LIN {X 101.722,Y -39.308,Z -42.456,A -90.000,B 90.000,C 0.000} C_DIS
LIN {X 102.625,Y -39.308,Z -41.468,A -90.000,B 90.000,C 0.000} C_DIS
LIN {X 103.587,Y -39.308,Z -40.444,A -90.000,B 90.000,C 0.000} C_DIS
LIN {X 104.451,Y -39.308,Z -39.577,A -90.000,B 90.000,C 0.000} C_DIS
LIN {X 104.780,Y -39.308,Z -39.269,A -90.000,B 90.000,C 0.000} C_DIS
LIN {X 105.201,Y -39.308,Z -38.850,A -90.000,B 90.000,C 0.000} C_DIS
LIN {X 105.598,Y -39.308,Z -38.492,A -90.000,B 90.000,C 0.000} C_DIS
LIN {X 106.174,Y -39.308,Z -37.998,A -90.000,B 90.000,C 0.000} C_DIS
LIN {X 106.785,Y -39.308,Z -37.546,A -90.000,B 90.000,C 0.000} C_DIS
LIN {X 107.016,Y -39.308,Z -37.381,A -90.000,B 90.000,C 0.000} C_DIS
LIN {X 107.121,Y -39.308,Z -37.313,A -90.000,B 90.000,C 0.000} C_DIS
LIN {X 107.510,Y -39.308,Z -37.082,A -90.000,B 90.000,C 0.000} C_DIS
LIN {X 107.952,Y -39.308,Z -36.851,A -90.000,B 90.000,C 0.000} C_DIS
LIN {X 108.136,Y -39.308,Z -36.762,A -90.000,B 90.000,C 0.000} C_DIS
LIN {X 108.391,Y -39.308,Z -36.644,A -90.000,B 90.000,C 0.000} C_DIS
LIN {X 109.204,Y -39.308,Z -36.354,A -90.000,B 90.000,C 0.000} C_DIS
LIN {X 109.672,Y -39.308,Z -36.239,A -90.000,B 90.000,C 0.000} C_DIS
LIN {X 109.904,Y -39.308,Z -36.196,A -90.000,B 90.000,C 0.000} C_DIS
LIN {X 110.509,Y -39.308,Z -36.111,A -90.000,B 90.000,C 0.000} C_DIS
LIN {X 110.992,Y -39.308,Z -36.094,A -90.000,B 90.000,C 0.000} C_DIS
LIN {X 111.151,Y -39.308,Z -36.098,A -90.000,B 90.000,C 0.000} C_DIS
LIN {X 111.344,Y -39.308,Z -36.107,A -90.000,B 90.000,C 0.000} C_DIS
LIN {X 111.775,Y -39.308,Z -36.137,A -90.000,B 90.000,C 0.000} C_DIS
LIN {X 112.250,Y -39.308,Z -36.219,A -90.000,B 90.000,C 0.000} C_DIS
LIN {X 112.476,Y -39.308,Z -36.273,A -90.000,B 90.000,C 0.000} C_DIS
LIN {X 112.642,Y -39.308,Z -36.317,A -90.000,B 90.000,C 0.000} C_DIS
LIN {X 112.938,Y -39.308,Z -36.401,A -90.000,B 90.000,C 0.000} C_DIS
LIN {X 113.127,Y -39.308,Z -36.468,A -90.000,B 90.000,C 0.000} C_DIS
LIN {X 113.176,Y -39.308,Z -36.483,A -90.000,B 90.000,C 0.000} C_DIS
LIN {X 113.621,Y -39.308,Z -36.653,A -90.000,B 90.000,C 0.000} C_DIS
LIN {X 113.933,Y -39.308,Z -36.809,A -90.000,B 90.000,C 0.000} C_DIS
LIN {X 114.096,Y -39.308,Z -36.887,A -90.000,B 90.000,C 0.000} C_DIS
LIN {X 114.199,Y -39.308,Z -36.943,A -90.000,B 90.000,C 0.000} C_DIS
LIN {X 114.406,Y -39.308,Z -37.049,A -90.000,B 90.000,C 0.000} C_DIS
LIN {X 114.803,Y -39.308,Z -37.294,A -90.000,B 90.000,C 0.000} C_DIS
LIN {X 115.172,Y -39.308,Z -37.581,A -90.000,B 90.000,C 0.000} C_DIS
LIN {X 115.508,Y -39.308,Z -37.906,A -90.000,B 90.000,C 0.000} C_DIS
LIN {X 115.807,Y -39.308,Z -38.265,A -90.000,B 90.000,C 0.000} C_DIS
LIN {X 116.012,Y -39.308,Z -38.542,A -90.000,B 90.000,C 0.000} C_DIS
LIN {X 116.272,Y -39.308,Z -38.931,A -90.000,B 90.000,C 0.000} C_DIS
LIN {X 116.488,Y -39.308,Z -39.345,A -90.000,B 90.000,C 0.000} C_DIS
LIN {X 116.814,Y -39.308,Z -40.176,A -90.000,B 90.000,C 0.000} C_DIS
LIN {X 116.939,Y -39.308,Z -40.634,A -90.000,B 90.000,C 0.000} C_DIS
LIN {X 117.006,Y -39.308,Z -40.932,A -90.000,B 90.000,C 0.000} C_DIS
LIN {X 117.081,Y -39.308,Z -41.395,A -90.000,B 90.000,C 0.000} C_DIS
LIN {X 117.103,Y -39.308,Z -41.641,A -90.000,B 90.000,C 0.000} C_DIS
LIN {X 117.128,Y -39.308,Z -42.111,A -90.000,B 90.000,C 0.000} C_DIS
LIN {X 117.128,Y -39.308,Z -42.230,A -90.000,B 90.000,C 0.000} C_DIS
LIN {X 117.115,Y -39.308,Z -42.566,A -90.000,B 90.000,C 0.000} C_DIS
LIN {X 117.020,Y -39.308,Z -43.281,A -90.000,B 90.000,C 0.000} C_DIS
LIN {X 116.910,Y -39.308,Z -43.735,A -90.000,B 90.000,C 0.000} C_DIS
LIN {X 116.846,Y -39.308,Z -43.965,A -90.000,B 90.000,C 0.000} C_DIS
LIN {X 116.721,Y -39.308,Z -44.363,A -90.000,B 90.000,C 0.000} C_DIS
LIN {X 116.671,Y -39.308,Z -44.527,A -90.000,B 90.000,C 0.000} C_DIS
LIN {X 116.543,Y -39.308,Z -44.969,A -90.000,B 90.000,C 0.000} C_DIS
LIN {X 116.287,Y -39.308,Z -45.797,A -90.000,B 90.000,C 0.000} C_DIS
LIN {X 116.068,Y -39.308,Z -46.437,A -90.000,B 90.000,C 0.000} C_DIS
LIN {X 115.942,Y -39.308,Z -46.787,A -90.000,B 90.000,C 0.000} C_DIS
LIN {X 115.595,Y -39.308,Z -47.692,A -90.000,B 90.000,C 0.000} C_DIS
LIN {X 115.490,Y -39.308,Z -47.931,A -90.000,B 90.000,C 0.000} C_DIS
LIN {X 115.109,Y -39.308,Z -48.763,A -90.000,B 90.000,C 0.000} C_DIS
LIN {X 114.640,Y -39.308,Z -49.738,A -90.000,B 90.000,C 0.000} C_DIS
LIN {X 114.310,Y -39.308,Z -50.406,A -90.000,B 90.000,C 0.000} C_DIS
LIN {X 113.759,Y -39.308,Z -51.507,A -90.000,B 90.000,C 0.000} C_DIS
LIN {X 113.170,Y -39.308,Z -52.723,A -90.000,B 90.000,C 0.000} C_DIS
LIN {X 112.487,Y -39.308,Z -54.223,A -90.000,B 90.000,C 0.000} C_DIS
LIN {X 112.277,Y -39.308,Z -54.728,A -90.000,B 90.000,C 0.000} C_DIS
LIN {X 111.817,Y -39.308,Z -55.818,A -90.000,B 90.000,C 0.000} C_DIS
LIN {X 111.518,Y -39.308,Z -56.593,A -90.000,B 90.000,C 0.000} C_DIS
LIN {X 111.203,Y -39.308,Z -57.396,A -90.000,B 90.000,C 0.000} C_DIS
LIN {X 110.924,Y -39.308,Z -58.174,A -90.000,B 90.000,C 0.000} C_DIS
LIN {X 110.658,Y -39.308,Z -58.905,A -90.000,B 90.000,C 0.000} C_DIS
LIN {X 109.994,Y -39.308,Z -60.877,A -90.000,B 90.000,C 0.000} C_DIS
LIN {X 109.296,Y -39.308,Z -62.984,A -90.000,B 90.000,C 0.000} C_DIS
LIN {X 108.534,Y -39.308,Z -65.215,A -90.000,B 90.000,C 0.000} C_DIS
LIN {X 107.818,Y -39.308,Z -67.178,A -90.000,B 90.000,C 0.000} C_DIS
LIN {X 107.521,Y -39.308,Z -67.986,A -90.000,B 90.000,C 0.000} C_DIS
LIN {X 106.574,Y -39.308,Z -70.314,A -90.000,B 90.000,C 0.000} C_DIS
LIN {X 106.354,Y -39.308,Z -70.809,A -90.000,B 90.000,C 0.000} C_DIS
LIN {X 105.509,Y -39.308,Z -72.687,A -90.000,B 90.000,C 0.000} C_DIS
LIN {X 105.305,Y -39.308,Z -73.108,A -90.000,B 90.000,C 0.000} C_DIS
LIN {X 104.664,Y -39.308,Z -74.413,A -90.000,B 90.000,C 0.000} C_DIS
LIN {X 104.177,Y -39.308,Z -75.400,A -90.000,B 90.000,C 0.000} C_DIS
LIN {X 103.035,Y -39.308,Z -77.509,A -90.000,B 90.000,C 0.000} C_DIS
LIN {X 102.762,Y -39.308,Z -77.959,A -90.000,B 90.000,C 0.000} C_DIS
LIN {X 102.514,Y -39.308,Z -78.356,A -90.000,B 90.000,C 0.000} C_DIS
LIN {X 101.738,Y -39.308,Z -79.581,A -90.000,B 90.000,C 0.000} C_DIS
LIN {X 101.385,Y -39.308,Z -80.081,A -90.000,B 90.000,C 0.000} C_DIS
LIN {X 100.588,Y -39.308,Z -81.180,A -90.000,B 90.000,C 0.000} C_DIS
LIN {X 100.385,Y -39.308,Z -81.459,A -90.000,B 90.000,C 0.000} C_DIS
LIN {X 99.790,Y -39.308,Z -82.216,A -90.000,B 90.000,C 0.000} C_DIS
LIN {X 99.306,Y -39.308,Z -82.840,A -90.000,B 90.000,C 0.000} C_DIS
LIN {X 99.040,Y -39.308,Z -83.162,A -90.000,B 90.000,C 0.000} C_DIS
LIN {X 98.410,Y -39.308,Z -83.929,A -90.000,B 90.000,C 0.000} C_DIS
LIN {X 98.289,Y -39.308,Z -84.069,A -90.000,B 90.000,C 0.000} C_DIS
LIN {X 97.421,Y -39.308,Z -85.030,A -90.000,B 90.000,C 0.000} C_DIS
LIN {X 96.998,Y -39.308,Z -85.453,A -90.000,B 90.000,C 0.000} C_DIS
LIN {X 96.306,Y -39.308,Z -86.108,A -90.000,B 90.000,C 0.000} C_DIS
LIN {X 96.127,Y -39.308,Z -86.274,A -90.000,B 90.000,C 0.000} C_DIS
LIN {X 95.588,Y -39.308,Z -86.759,A -90.000,B 90.000,C 0.000} C_DIS
LIN {X 94.996,Y -39.308,Z -87.295,A -90.000,B 90.000,C 0.000} C_DIS
LIN {X 94.639,Y -39.308,Z -87.627,A -90.000,B 90.000,C 0.000} C_DIS
LIN {X 94.383,Y -39.308,Z -87.833,A -90.000,B 90.000,C 0.000} C_DIS
LIN {X 94.053,Y -39.308,Z -88.118,A -90.000,B 90.000,C 0.000} C_DIS
LIN {X 93.745,Y -39.308,Z -88.370,A -90.000,B 90.000,C 0.000} C_DIS
LIN {X 93.562,Y -39.308,Z -88.554,A -90.000,B 90.000,C 0.000} C_DIS
LIN {X 93.370,Y -39.308,Z -88.839,A -90.000,B 90.000,C 0.000} C_DIS
LIN {X 93.332,Y -39.308,Z -88.909,A -90.000,B 90.000,C 0.000} C_DIS
LIN {X 93.219,Y -39.308,Z -89.185,A -90.000,B 90.000,C 0.000} C_DIS
LIN {X 93.090,Y -39.308,Z -89.585,A -90.000,B 90.000,C 0.000} C_DIS
LIN {X 92.874,Y -39.308,Z -90.727,A -90.000,B 90.000,C 0.000} C_DIS
LIN {X 92.802,Y -39.308,Z -91.038,A -90.000,B 90.000,C 0.000} C_DIS
LIN {X 92.618,Y -39.308,Z -92.389,A -90.000,B 90.000,C 0.000} C_DIS
LIN {X 92.595,Y -39.308,Z -92.544,A -90.000,B 90.000,C 0.000} C_DIS
LIN {X 92.499,Y -39.308,Z -93.287,A -90.000,B 90.000,C 0.000} C_DIS
LIN {X 92.352,Y -39.308,Z -94.370,A -90.000,B 90.000,C 0.000} C_DIS
LIN {X 92.295,Y -39.308,Z -94.744,A -90.000,B 90.000,C 0.000} C_DIS
LIN {X 92.054,Y -39.308,Z -96.144,A -90.000,B 90.000,C 0.000} C_DIS
LIN {X 91.937,Y -39.308,Z -96.559,A -90.000,B 90.000,C 0.000} C_DIS
LIN {X 91.815,Y -39.308,Z -96.959,A -90.000,B 90.000,C 0.000} C_DIS
LIN {X 91.618,Y -39.308,Z -97.654,A -90.000,B 90.000,C 0.000} C_DIS
LIN {X 91.465,Y -39.308,Z -98.026,A -90.000,B 90.000,C 0.000} C_DIS
LIN {X 91.067,Y -39.308,Z -98.874,A -90.000,B 90.000,C 0.000} C_DIS
LIN {X 90.869,Y -39.308,Z -99.224,A -90.000,B 90.000,C 0.000} C_DIS
LIN {X 90.401,Y -39.308,Z -99.888,A -90.000,B 90.000,C 0.000} C_DIS
LIN {X 89.790,Y -39.308,Z -100.675,A -90.000,B 90.000,C 0.000} C_DIS
LIN {X 89.275,Y -39.308,Z -101.469,A -90.000,B 90.000,C 0.000} C_DIS
LIN {X 88.799,Y -39.308,Z -102.371,A -90.000,B 90.000,C 0.000} C_DIS
LIN {X 88.475,Y -39.308,Z -103.161,A -90.000,B 90.000,C 0.000} C_DIS
LIN {X 88.332,Y -39.308,Z -103.810,A -90.000,B 90.000,C 0.000} C_DIS
LIN {X 88.359,Y -39.308,Z -104.371,A -90.000,B 90.000,C 0.000} C_DIS
LIN {X 88.567,Y -39.308,Z -105.406,A -90.000,B 90.000,C 0.000} C_DIS
LIN {X 88.806,Y -39.308,Z -106.627,A -90.000,B 90.000,C 0.000} C_DIS
LIN {X 88.934,Y -39.308,Z -108.256,A -90.000,B 90.000,C 0.000} C_DIS
LIN {X 88.949,Y -39.308,Z -108.491,A -90.000,B 90.000,C 0.000} C_DIS
LIN {X 88.942,Y -39.308,Z -108.668,A -90.000,B 90.000,C 0.000} C_DIS
LIN {X 88.800,Y -39.308,Z -110.495,A -90.000,B 90.000,C 0.000} C_DIS
LIN {X 88.774,Y -39.308,Z -110.765,A -90.000,B 90.000,C 0.000} C_DIS
LIN {X 88.667,Y -39.308,Z -111.550,A -90.000,B 90.000,C 0.000} C_DIS
LIN {X 88.430,Y -39.308,Z -112.947,A -90.000,B 90.000,C 0.000} C_DIS
LIN {X 88.207,Y -39.308,Z -114.211,A -90.000,B 90.000,C 0.000} C_DIS
LIN {X 87.996,Y -39.308,Z -115.227,A -90.000,B 90.000,C 0.000} C_DIS
LIN {X 87.956,Y -39.308,Z -115.438,A -90.000,B 90.000,C 0.000} C_DIS
LIN {X 87.638,Y -39.308,Z -117.389,A -90.000,B 90.000,C 0.000} C_DIS
LIN {X 87.573,Y -39.308,Z -118.816,A -90.000,B 90.000,C 0.000} C_DIS
LIN {X 87.557,Y -39.308,Z -119.381,A -90.000,B 90.000,C 0.000} C_DIS
LIN {X 87.603,Y -39.308,Z -120.775,A -90.000,B 90.000,C 0.000} C_DIS
LIN {X 87.657,Y -39.308,Z -121.429,A -90.000,B 90.000,C 0.000} C_DIS
LIN {X 87.731,Y -39.308,Z -122.583,A -90.000,B 90.000,C 0.000} C_DIS
LIN {X 87.800,Y -39.308,Z -123.097,A -90.000,B 90.000,C 0.000} C_DIS
LIN {X 87.825,Y -39.308,Z -123.409,A -90.000,B 90.000,C 0.000} C_DIS
LIN {X 87.876,Y -39.308,Z -124.655,A -90.000,B 90.000,C 0.000} C_DIS
LIN {X 87.918,Y -39.308,Z -125.034,A -90.000,B 90.000,C 0.000} C_DIS
LIN {X 87.941,Y -39.308,Z -125.333,A -90.000,B 90.000,C 0.000} C_DIS
LIN {X 87.951,Y -39.308,Z -125.837,A -90.000,B 90.000,C 0.000} C_DIS
LIN {X 87.901,Y -39.308,Z -127.285,A -90.000,B 90.000,C 0.000} C_DIS
LIN {X 87.877,Y -39.308,Z -127.831,A -90.000,B 90.000,C 0.000} C_DIS
LIN {X 87.851,Y -39.308,Z -128.184,A -90.000,B 90.000,C 0.000} C_DIS
LIN {X 87.757,Y -39.308,Z -129.307,A -90.000,B 90.000,C 0.000} C_DIS
LIN {X 87.684,Y -39.308,Z -130.314,A -90.000,B 90.000,C 0.000} C_DIS
LIN {X 87.557,Y -39.308,Z -131.579,A -90.000,B 90.000,C 0.000} C_DIS
LIN {X 87.475,Y -39.308,Z -132.714,A -90.000,B 90.000,C 0.000} C_DIS
LIN {X 87.343,Y -39.308,Z -134.110,A -90.000,B 90.000,C 0.000} C_DIS
LIN {X 87.221,Y -39.308,Z -135.777,A -90.000,B 90.000,C 0.000} C_DIS
LIN {X 87.144,Y -39.308,Z -137.172,A -90.000,B 90.000,C 0.000} C_DIS
LIN {X 87.005,Y -39.308,Z -139.170,A -90.000,B 90.000,C 0.000} C_DIS
LIN {X 86.928,Y -39.308,Z -140.602,A -90.000,B 90.000,C 0.000} C_DIS
LIN {X 86.747,Y -39.308,Z -142.945,A -90.000,B 90.000,C 0.000} C_DIS
LIN {X 86.662,Y -39.308,Z -144.278,A -90.000,B 90.000,C 0.000} C_DIS
LIN {X 86.407,Y -39.308,Z -146.950,A -90.000,B 90.000,C 0.000} C_DIS
LIN {X 86.303,Y -39.308,Z -148.174,A -90.000,B 90.000,C 0.000} C_DIS
LIN {X 86.278,Y -39.308,Z -148.428,A -90.000,B 90.000,C 0.000} C_DIS
LIN {X 86.171,Y -39.308,Z -149.383,A -90.000,B 90.000,C 0.000} C_DIS
LIN {X 85.816,Y -39.308,Z -152.222,A -90.000,B 90.000,C 0.000} C_DIS
LIN {X 85.710,Y -39.308,Z -152.942,A -90.000,B 90.000,C 0.000} C_DIS
LIN {X 85.232,Y -39.308,Z -155.979,A -90.000,B 90.000,C 0.000} C_DIS
LIN {X 85.136,Y -39.308,Z -156.498,A -90.000,B 90.000,C 0.000} C_DIS
LIN {X 84.520,Y -39.308,Z -159.679,A -90.000,B 90.000,C 0.000} C_DIS
LIN {X 84.432,Y -39.308,Z -160.063,A -90.000,B 90.000,C 0.000} C_DIS
LIN {X 83.664,Y -39.308,Z -163.335,A -90.000,B 90.000,C 0.000} C_DIS
LIN {X 83.589,Y -39.308,Z -163.643,A -90.000,B 90.000,C 0.000} C_DIS
LIN {X 82.601,Y -39.308,Z -167.169,A -90.000,B 90.000,C 0.000} C_DIS
LIN {X 81.544,Y -39.308,Z -170.573,A -90.000,B 90.000,C 0.000} C_DIS
LIN {X 80.492,Y -39.308,Z -173.831,A -90.000,B 90.000,C 0.000} C_DIS
LIN {X 80.289,Y -39.308,Z -174.485,A -90.000,B 90.000,C 0.000} C_DIS
LIN {X 79.518,Y -39.308,Z -176.924,A -90.000,B 90.000,C 0.000} C_DIS
LIN {X 78.896,Y -39.308,Z -179.083,A -90.000,B 90.000,C 0.000} C_DIS
LIN {X 78.733,Y -39.308,Z -179.680,A -90.000,B 90.000,C 0.000} C_DIS
LIN {X 78.239,Y -39.308,Z -181.531,A -90.000,B 90.000,C 0.000} C_DIS
LIN {X 78.020,Y -39.308,Z -182.417,A -90.000,B 90.000,C 0.000} C_DIS
LIN {X 77.515,Y -39.308,Z -184.388,A -90.000,B 90.000,C 0.000} C_DIS
LIN {X 77.360,Y -39.308,Z -185.055,A -90.000,B 90.000,C 0.000} C_DIS
LIN {X 76.824,Y -39.308,Z -187.147,A -90.000,B 90.000,C 0.000} C_DIS
LIN {X 76.720,Y -39.308,Z -187.594,A -90.000,B 90.000,C 0.000} C_DIS
LIN {X 76.130,Y -39.308,Z -189.797,A -90.000,B 90.000,C 0.000} C_DIS
LIN {X 76.066,Y -39.308,Z -190.059,A -90.000,B 90.000,C 0.000} C_DIS
LIN {X 75.356,Y -39.308,Z -192.504,A -90.000,B 90.000,C 0.000} C_DIS
LIN {X 75.319,Y -39.308,Z -192.641,A -90.000,B 90.000,C 0.000} C_DIS
LIN {X 75.217,Y -39.308,Z -192.988,A -90.000,B 90.000,C 0.000} C_DIS
LIN {X 74.311,Y -39.308,Z -195.828,A -90.000,B 90.000,C 0.000} C_DIS
LIN {X 73.163,Y -39.308,Z -199.116,A -90.000,B 90.000,C 0.000} C_DIS
LIN {X 71.708,Y -39.308,Z -203.024,A -90.000,B 90.000,C 0.000} C_DIS
LIN {X 69.982,Y -39.308,Z -207.432,A -90.000,B 90.000,C 0.000} C_DIS
LIN {X 67.893,Y -39.308,Z -212.535,A -90.000,B 90.000,C 0.000} C_DIS
LIN {X 66.291,Y -39.308,Z -216.289,A -90.000,B 90.000,C 0.000} C_DIS
LIN {X 65.715,Y -39.308,Z -217.628,A -90.000,B 90.000,C 0.000} C_DIS
LIN {X 63.402,Y -39.308,Z -222.773,A -90.000,B 90.000,C 0.000} C_DIS
LIN {X 60.817,Y -39.308,Z -228.203,A -90.000,B 90.000,C 0.000} C_DIS
LIN {X 58.290,Y -39.308,Z -233.168,A -90.000,B 90.000,C 0.000} C_DIS
LIN {X 58.161,Y -39.308,Z -233.430,A -90.000,B 90.000,C 0.000} C_DIS
LIN {X 58.084,Y -39.308,Z -233.572,A -90.000,B 90.000,C 0.000} C_DIS
LIN {X 55.501,Y -39.308,Z -238.273,A -90.000,B 90.000,C 0.000} C_DIS
LIN {X 55.234,Y -39.308,Z -238.790,A -90.000,B 90.000,C 0.000} C_DIS
LIN {X 54.905,Y -39.308,Z -239.394,A -90.000,B 90.000,C 0.000} C_DIS
LIN {X 54.713,Y -39.308,Z -239.734,A -90.000,B 90.000,C 0.000} C_DIS
LIN {X 52.416,Y -39.308,Z -243.561,A -90.000,B 90.000,C 0.000} C_DIS
LIN {X 52.416,Y -60.000,Z -243.561,A -90.000,B 90.000,C 0.000} C_DIS
LIN {X 101.612,Y -60.000,Z -42.574,A -90.000,B 90.000,C 0.000} C_DIS
LIN {X 101.612,Y -37.308,Z -42.574,A -90.000,B 90.000,C 0.000} C_DIS
LIN {X 101.629,Y -37.311,Z -42.419,A -90.000,B 90.000,C 0.000} C_DIS
LIN {X 101.656,Y -37.315,Z -42.297,A -90.000,B 90.000,C 0.000} C_DIS
LIN {X 101.723,Y -37.329,Z -42.033,A -90.000,B 90.000,C 0.000} C_DIS
LIN {X 101.775,Y -37.337,Z -41.902,A -90.000,B 90.000,C 0.000} C_DIS
LIN {X 101.877,Y -37.355,Z -41.654,A -90.000,B 90.000,C 0.000} C_DIS
LIN {X 102.047,Y -37.380,Z -41.312,A -90.000,B 90.000,C 0.000} C_DIS
LIN {X 102.134,Y -37.395,Z -41.144,A -90.000,B 90.000,C 0.000} C_DIS
LIN {X 102.399,Y -37.434,Z -40.690,A -90.000,B 90.000,C 0.000} C_DIS
LIN {X 102.645,Y -37.468,Z -40.302,A -90.000,B 90.000,C 0.000} C_DIS
LIN {X 102.898,Y -37.488,Z -39.967,A -90.000,B 90.000,C 0.000} C_DIS
LIN {X 103.145,Y -37.508,Z -39.654,A -90.000,B 90.000,C 0.000} C_DIS
LIN {X 103.251,Y -37.517,Z -39.521,A -90.000,B 90.000,C 0.000} C_DIS
LIN {X 103.626,Y -37.529,Z -39.112,A -90.000,B 90.000,C 0.000} C_DIS
LIN {X 103.738,Y -37.531,Z -38.993,A -90.000,B 90.000,C 0.000} C_DIS
LIN {X 103.970,Y -37.536,Z -38.759,A -90.000,B 90.000,C 0.000} C_DIS
LIN {X 104.139,Y -37.537,Z -38.598,A -90.000,B 90.000,C 0.000} C_DIS
LIN {X 104.427,Y -37.532,Z -38.323,A -90.000,B 90.000,C 0.000} C_DIS
LIN {X 104.582,Y -37.527,Z -38.183,A -90.000,B 90.000,C 0.000} C_DIS
LIN {X 104.958,Y -37.514,Z -37.880,A -90.000,B 90.000,C 0.000} C_DIS
LIN {X 105.114,Y -37.508,Z -37.759,A -90.000,B 90.000,C 0.000} C_DIS
LIN {X 105.454,Y -37.493,Z -37.511,A -90.000,B 90.000,C 0.000} C_DIS
LIN {X 105.665,Y -37.480,Z -37.367,A -90.000,B 90.000,C 0.000} C_DIS
LIN {X 105.896,Y -37.473,Z -37.215,A -90.000,B 90.000,C 0.000} C_DIS
LIN {X 106.119,Y -37.463,Z -37.081,A -90.000,B 90.000,C 0.000} C_DIS
LIN {X 106.362,Y -37.448,Z -36.944,A -90.000,B 90.000,C 0.000} C_DIS
LIN {X 106.738,Y -37.432,Z -36.736,A -90.000,B 90.000,C 0.000} C_DIS
LIN {X 106.867,Y -37.429,Z -36.668,A -90.000,B 90.000,C 0.000} C_DIS
LIN {X 106.984,Y -37.425,Z -36.612,A -90.000,B 90.000,C 0.000} C_DIS
LIN {X 107.278,Y -37.416,Z -36.473,A -90.000,B 90.000,C 0.000} C_DIS
LIN {X 107.430,Y -37.413,Z -36.403,A -90.000,B 90.000,C 0.000} C_DIS
LIN {X 107.770,Y -37.406,Z -36.252,A -90.000,B 90.000,C 0.000} C_DIS
LIN {X 108.143,Y -37.398,Z -36.107,A -90.000,B 90.000,C 0.000} C_DIS
LIN {X 108.234,Y -37.397,Z -36.075,A -90.000,B 90.000,C 0.000} C_DIS
LIN {X 108.294,Y -37.398,Z -36.051,A -90.000,B 90.000,C 0.000} C_DIS
LIN {X 109.071,Y -37.390,Z -35.804,A -90.000,B 90.000,C 0.000} C_DIS
LIN {X 109.166,Y -37.391,Z -35.777,A -90.000,B 90.000,C 0.000} C_DIS
LIN {X 109.380,Y -37.390,Z -35.728,A -90.000,B 90.000,C 0.000} C_DIS
LIN {X 109.499,Y -37.389,Z -35.704,A -90.000,B 90.000,C 0.000} C_DIS
LIN {X 109.570,Y -37.389,Z -35.688,A -90.000,B 90.000,C 0.000} C_DIS
LIN {X 109.857,Y -37.390,Z -35.632,A -90.000,B 90.000,C 0.000} C_DIS
LIN {X 110.012,Y -37.392,Z -35.602,A -90.000,B 90.000,C 0.000} C_DIS
LIN {X 110.069,Y -37.392,Z -35.595,A -90.000,B 90.000,C 0.000} C_DIS
LIN {X 110.465,Y -37.387,Z -35.558,A -90.000,B 90.000,C 0.000} C_DIS
LIN {X 111.003,Y -37.390,Z -35.530,A -90.000,B 90.000,C 0.000} C_DIS
LIN {X 111.317,Y -37.391,Z -35.537,A -90.000,B 90.000,C 0.000} C_DIS
LIN {X 111.666,Y -37.392,Z -35.557,A -90.000,B 90.000,C 0.000} C_DIS
LIN {X 111.823,Y -37.390,Z -35.574,A -90.000,B 90.000,C 0.000} C_DIS
LIN {X 112.066,Y -37.392,Z -35.605,A -90.000,B 90.000,C 0.000} C_DIS
LIN {X 112.386,Y -37.394,Z -35.655,A -90.000,B 90.000,C 0.000} C_DIS
LIN {X 112.546,Y -37.398,Z -35.681,A -90.000,B 90.000,C 0.000} C_DIS
LIN {X 112.867,Y -37.398,Z -35.764,A -90.000,B 90.000,C 0.000} C_DIS
LIN {X 113.101,Y -37.399,Z -35.828,A -90.000,B 90.000,C 0.000} C_DIS
LIN {X 113.182,Y -37.400,Z -35.851,A -90.000,B 90.000,C 0.000} C_DIS
LIN {X 113.401,Y -37.401,Z -35.926,A -90.000,B 90.000,C 0.000} C_DIS
LIN {X 113.848,Y -37.399,Z -36.104,A -90.000,B 90.000,C 0.000} C_DIS
LIN {X 114.023,Y -37.401,Z -36.180,A -90.000,B 90.000,C 0.000} C_DIS
LIN {X 114.165,Y -37.404,Z -36.241,A -90.000,B 90.000,C 0.000} C_DIS
LIN {X 114.592,Y -37.402,Z -36.465,A -90.000,B 90.000,C 0.000} C_DIS
LIN {X 114.656,Y -37.401,Z -36.500,A -90.000,B 90.000,C 0.000} C_DIS
LIN {X 115.108,Y -37.394,Z -36.801,A -90.000,B 90.000,C 0.000} C_DIS
LIN {X 115.164,Y -37.394,Z -36.841,A -90.000,B 90.000,C 0.000} C_DIS
LIN {X 115.527,Y -37.390,Z -37.143,A -90.000,B 90.000,C 0.000} C_DIS
LIN {X 115.726,Y -37.387,Z -37.344,A -90.000,B 90.000,C 0.000} C_DIS
LIN {X 115.932,Y -37.385,Z -37.557,A -90.000,B 90.000,C 0.000} C_DIS
LIN {X 116.140,Y -37.386,Z -37.800,A -90.000,B 90.000,C 0.000} C_DIS
LIN {X 116.249,Y -37.385,Z -37.938,A -90.000,B 90.000,C 0.000} C_DIS
LIN {X 116.441,Y -37.388,Z -38.181,A -90.000,B 90.000,C 0.000} C_DIS
LIN {X 116.702,Y -37.384,Z -38.591,A -90.000,B 90.000,C 0.000} C_DIS
LIN {X 116.836,Y -37.381,Z -38.860,A -90.000,B 90.000,C 0.000} C_DIS
LIN {X 116.930,Y -37.379,Z -39.049,A -90.000,B 90.000,C 0.000} C_DIS
LIN {X 116.972,Y -37.377,Z -39.155,A -90.000,B 90.000,C 0.000} C_DIS
LIN {X 117.070,Y -37.377,Z -39.405,A -90.000,B 90.000,C 0.000} C_DIS
LIN {X 117.242,Y -37.375,Z -39.860,A -90.000,B 90.000,C 0.000} C_DIS
LIN {X 117.288,Y -37.371,Z -40.034,A -90.000,B 90.000,C 0.000} C_DIS
LIN {X 117.365,Y -37.370,Z -40.328,A -90.000,B 90.000,C 0.000} C_DIS
LIN {X 117.387,Y -37.368,Z -40.432,A -90.000,B 90.000,C 0.000} C_DIS
LIN {X 117.421,Y -37.365,Z -40.627,A -90.000,B 90.000,C 0.000} C_DIS
LIN {X 117.443,Y -37.365,Z -40.728,A -90.000,B 90.000,C 0.000} C_DIS
LIN {X 117.518,Y -37.362,Z -41.208,A -90.000,B 90.000,C 0.000} C_DIS
LIN {X 117.529,Y -37.361,Z -41.323,A -90.000,B 90.000,C 0.000} C_DIS
LIN {X 117.541,Y -37.361,Z -41.406,A -90.000,B 90.000,C 0.000} C_DIS
LIN {X 117.552,Y -37.362,Z -41.518,A -90.000,B 90.000,C 0.000} C_DIS
LIN {X 117.566,Y -37.363,Z -41.618,A -90.000,B 90.000,C 0.000} C_DIS
LIN {X 117.582,Y -37.364,Z -41.824,A -90.000,B 90.000,C 0.000} C_DIS
LIN {X 117.598,Y -37.364,Z -42.113,A -90.000,B 90.000,C 0.000} C_DIS
LIN {X 117.615,Y -37.371,Z -42.456,A -90.000,B 90.000,C 0.000} C_DIS
LIN {X 117.612,Y -37.371,Z -42.585,A -90.000,B 90.000,C 0.000} C_DIS
LIN {X 117.603,Y -37.375,Z -42.769,A -90.000,B 90.000,C 0.000} C_DIS
LIN {X 117.568,Y -37.384,Z -43.280,A -90.000,B 90.000,C 0.000} C_DIS
LIN {X 117.546,Y -37.385,Z -43.434,A -90.000,B 90.000,C 0.000} C_DIS
LIN {X 117.522,Y -37.389,Z -43.592,A -90.000,B 90.000,C 0.000} C_DIS
LIN {X 117.495,Y -37.396,Z -43.809,A -90.000,B 90.000,C 0.000} C_DIS
LIN {X 117.421,Y -37.410,Z -44.234,A -90.000,B 90.000,C 0.000} C_DIS
LIN {X 117.382,Y -37.415,Z -44.407,A -90.000,B 90.000,C 0.000} C_DIS
LIN {X 117.286,Y -37.424,Z -44.814,A -90.000,B 90.000,C 0.000} C_DIS
LIN {X 117.193,Y -37.430,Z -45.193,A -90.000,B 90.000,C 0.000} C_DIS
LIN {X 117.168,Y -37.432,Z -45.287,A -90.000,B 90.000,C 0.000} C_DIS
LIN {X 116.978,Y -37.434,Z -45.926,A -90.000,B 90.000,C 0.000} C_DIS
LIN {X 116.921,Y -37.433,Z -46.095,A -90.000,B 90.000,C 0.000} C_DIS
LIN {X 116.602,Y -37.428,Z -46.967,A -90.000,B 90.000,C 0.000} C_DIS
LIN {X 116.539,Y -37.429,Z -47.137,A -90.000,B 90.000,C 0.000} C_DIS
LIN {X 116.189,Y -37.416,Z -47.952,A -90.000,B 90.000,C 0.000} C_DIS
LIN {X 116.156,Y -37.416,Z -48.026,A -90.000,B 90.000,C 0.000} C_DIS
LIN {X 115.889,Y -37.410,Z -48.572,A -90.000,B 90.000,C 0.000} C_DIS
LIN {X 115.501,Y -37.403,Z -49.350,A -90.000,B 90.000,C 0.000} C_DIS
LIN {X 115.430,Y -37.402,Z -49.492,A -90.000,B 90.000,C 0.000} C_DIS
LIN {X 114.861,Y -37.394,Z -50.596,A -90.000,B 90.000,C 0.000} C_DIS
LIN {X 114.199,Y -37.389,Z -51.887,A -90.000,B 90.000,C 0.000} C_DIS
LIN {X 113.591,Y -37.385,Z -53.125,A -90.000,B 90.000,C 0.000} C_DIS
LIN {X 113.530,Y -37.385,Z -53.256,A -90.000,B 90.000,C 0.000} C_DIS
LIN {X 113.048,Y -37.385,Z -54.319,A -90.000,B 90.000,C 0.000} C_DIS
LIN {X 112.975,Y -37.387,Z -54.492,A -90.000,B 90.000,C 0.000} C_DIS
LIN {X 112.392,Y -37.388,Z -55.887,A -90.000,B 90.000,C 0.000} C_DIS
LIN {X 111.753,Y -37.390,Z -57.546,A -90.000,B 90.000,C 0.000} C_DIS
LIN {X 111.203,Y -37.393,Z -59.096,A -90.000,B 90.000,C 0.000} C_DIS
LIN {X 110.557,Y -37.398,Z -61.065,A -90.000,B 90.000,C 0.000} C_DIS
LIN {X 109.947,Y -37.403,Z -62.950,A -90.000,B 90.000,C 0.000} C_DIS
LIN {X 109.226,Y -37.404,Z -65.082,A -90.000,B 90.000,C 0.000} C_DIS
LIN {X 108.967,Y -37.403,Z -65.799,A -90.000,B 90.000,C 0.000} C_DIS
LIN {X 108.309,Y -37.403,Z -67.604,A -90.000,B 90.000,C 0.000} C_DIS
LIN {X 108.225,Y -37.403,Z -67.833,A -90.000,B 90.000,C 0.000} C_DIS
LIN {X 108.076,Y -37.400,Z -68.212,A -90.000,B 90.000,C 0.000} C_DIS
LIN {X 107.446,Y -37.404,Z -69.796,A -90.000,B 90.000,C 0.000} C_DIS
LIN {X 107.263,Y -37.405,Z -70.252,A -90.000,B 90.000,C 0.000} C_DIS
LIN {X 107.131,Y -37.403,Z -70.562,A -90.000,B 90.000,C 0.000} C_DIS
LIN {X 106.480,Y -37.411,Z -72.071,A -90.000,B 90.000,C 0.000} C_DIS
LIN {X 106.196,Y -37.413,Z -72.716,A -90.000,B 90.000,C 0.000} C_DIS
LIN {X 105.877,Y -37.413,Z -73.388,A -90.000,B 90.000,C 0.000} C_DIS
LIN {X 105.250,Y -37.419,Z -74.707,A -90.000,B 90.000,C 0.000} C_DIS
LIN {X 105.072,Y -37.421,Z -75.080,A -90.000,B 90.000,C 0.000} C_DIS
LIN {X 104.900,Y -37.421,Z -75.429,A -90.000,B 90.000,C 0.000} C_DIS
LIN {X 104.753,Y -37.419,Z -75.712,A -90.000,B 90.000,C 0.000} C_DIS
LIN {X 104.386,Y -37.423,Z -76.414,A -90.000,B 90.000,C 0.000} C_DIS
LIN {X 103.785,Y -37.431,Z -77.572,A -90.000,B 90.000,C 0.000} C_DIS
LIN {X 103.595,Y -37.428,Z -77.899,A -90.000,B 90.000,C 0.000} C_DIS
LIN {X 103.168,Y -37.435,Z -78.630,A -90.000,B 90.000,C 0.000} C_DIS
LIN {X 102.802,Y -37.445,Z -79.256,A -90.000,B 90.000,C 0.000} C_DIS
LIN {X 102.670,Y -37.446,Z -79.472,A -90.000,B 90.000,C 0.000} C_DIS
LIN {X 102.431,Y -37.446,Z -79.850,A -90.000,B 90.000,C 0.000} C_DIS
LIN {X 102.263,Y -37.446,Z -80.100,A -90.000,B 90.000,C 0.000} C_DIS
LIN {X 101.641,Y -37.458,Z -81.020,A -90.000,B 90.000,C 0.000} C_DIS
LIN {X 101.342,Y -37.466,Z -81.465,A -90.000,B 90.000,C 0.000} C_DIS
LIN {X 100.998,Y -37.466,Z -81.940,A -90.000,B 90.000,C 0.000} C_DIS
LIN {X 100.316,Y -37.486,Z -82.881,A -90.000,B 90.000,C 0.000} C_DIS
LIN {X 99.946,Y -37.489,Z -83.371,A -90.000,B 90.000,C 0.000} C_DIS
LIN {X 99.578,Y -37.501,Z -83.856,A -90.000,B 90.000,C 0.000} C_DIS
LIN {X 99.261,Y -37.508,Z -84.264,A -90.000,B 90.000,C 0.000} C_DIS
LIN {X 99.033,Y -37.512,Z -84.555,A -90.000,B 90.000,C 0.000} C_DIS
LIN {X 98.364,Y -37.544,Z -85.391,A -90.000,B 90.000,C 0.000} C_DIS
LIN {X 98.095,Y -37.550,Z -85.703,A -90.000,B 90.000,C 0.000} C_DIS
LIN {X 97.667,Y -37.573,Z -86.186,A -90.000,B 90.000,C 0.000} C_DIS
LIN {X 97.025,Y -37.612,Z -86.887,A -90.000,B 90.000,C 0.000} C_DIS
LIN {X 96.296,Y -37.671,Z -87.668,A -90.000,B 90.000,C 0.000} C_DIS
LIN {X 96.049,Y -37.693,Z -87.933,A -90.000,B 90.000,C 0.000} C_DIS
LIN {X 95.768,Y -37.712,Z -88.223,A -90.000,B 90.000,C 0.000} C_DIS
LIN {X 95.527,Y -37.724,Z -88.468,A -90.000,B 90.000,C 0.000} C_DIS
LIN {X 95.414,Y -37.740,Z -88.596,A -90.000,B 90.000,C 0.000} C_DIS
LIN {X 95.283,Y -37.762,Z -88.737,A -90.000,B 90.000,C 0.000} C_DIS
LIN {X 95.137,Y -37.809,Z -88.930,A -90.000,B 90.000,C 0.000} C_DIS
LIN {X 95.057,Y -37.828,Z -89.028,A -90.000,B 90.000,C 0.000} C_DIS
LIN {X 94.951,Y -37.875,Z -89.185,A -90.000,B 90.000,C 0.000} C_DIS
LIN {X 94.862,Y -37.915,Z -89.309,A -90.000,B 90.000,C 0.000} C_DIS
LIN {X 94.745,Y -37.967,Z -89.468,A -90.000,B 90.000,C 0.000} C_DIS
LIN {X 94.719,Y -37.976,Z -89.506,A -90.000,B 90.000,C 0.000} C_DIS
LIN {X 94.678,Y -37.988,Z -89.586,A -90.000,B 90.000,C 0.000} C_DIS
LIN {X 94.654,Y -37.992,Z -89.654,A -90.000,B 90.000,C 0.000} C_DIS
LIN {X 94.638,Y -37.996,Z -89.703,A -90.000,B 90.000,C 0.000} C_DIS
LIN {X 94.564,Y -38.006,Z -89.961,A -90.000,B 90.000,C 0.000} C_DIS
LIN {X 94.501,Y -37.998,Z -90.254,A -90.000,B 90.000,C 0.000} C_DIS
LIN {X 94.353,Y -37.992,Z -91.007,A -90.000,B 90.000,C 0.000} C_DIS
LIN {X 94.290,Y -37.999,Z -91.311,A -90.000,B 90.000,C 0.000} C_DIS
LIN {X 94.101,Y -37.984,Z -92.611,A -90.000,B 90.000,C 0.000} C_DIS
LIN {X 94.070,Y -37.984,Z -92.818,A -90.000,B 90.000,C 0.000} C_DIS
LIN {X 93.913,Y -37.974,Z -93.948,A -90.000,B 90.000,C 0.000} C_DIS
LIN {X 93.822,Y -37.971,Z -94.588,A -90.000,B 90.000,C 0.000} C_DIS
LIN {X 93.755,Y -37.965,Z -94.995,A -90.000,B 90.000,C 0.000} C_DIS
LIN {X 93.555,Y -37.959,Z -96.126,A -90.000,B 90.000,C 0.000} C_DIS
LIN {X 93.490,Y -37.944,Z -96.420,A -90.000,B 90.000,C 0.000} C_DIS
LIN {X 93.467,Y -37.942,Z -96.514,A -90.000,B 90.000,C 0.000} C_DIS
LIN {X 93.333,Y -37.941,Z -96.985,A -90.000,B 90.000,C 0.000} C_DIS
LIN {X 93.225,Y -37.947,Z -97.360,A -90.000,B 90.000,C 0.000} C_DIS
LIN {X 93.161,Y -37.949,Z -97.590,A -90.000,B 90.000,C 0.000} C_DIS
LIN {X 93.065,Y -37.941,Z -97.900,A -90.000,B 90.000,C 0.000} C_DIS
LIN {X 93.052,Y -37.940,Z -97.943,A -90.000,B 90.000,C 0.000} C_DIS
LIN {X 92.986,Y -37.928,Z -98.127,A -90.000,B 90.000,C 0.000} C_DIS
LIN {X 92.880,Y -37.928,Z -98.391,A -90.000,B 90.000,C 0.000} C_DIS
LIN {X 92.777,Y -37.930,Z -98.642,A -90.000,B 90.000,C 0.000} C_DIS
LIN {X 92.700,Y -37.936,Z -98.819,A -90.000,B 90.000,C 0.000} C_DIS
LIN {X 92.504,Y -37.935,Z -99.235,A -90.000,B 90.000,C 0.000} C_DIS
LIN {X 92.382,Y -37.923,Z -99.469,A -90.000,B 90.000,C 0.000} C_DIS
LIN {X 92.331,Y -37.921,Z -99.562,A -90.000,B 90.000,C 0.000} C_DIS
LIN {X 92.130,Y -37.919,Z -99.915,A -90.000,B 90.000,C 0.000} C_DIS
LIN {X 92.056,Y -37.921,Z -100.038,A -90.000,B 90.000,C 0.000} C_DIS
LIN {X 91.988,Y -37.926,Z -100.144,A -90.000,B 90.000,C 0.000} C_DIS
LIN {X 91.563,Y -37.946,Z -100.779,A -90.000,B 90.000,C 0.000} C_DIS
LIN {X 91.542,Y -37.948,Z -100.808,A -90.000,B 90.000,C 0.000} C_DIS
LIN {X 91.031,Y -38.022,Z -101.576,A -90.000,B 90.000,C 0.000} C_DIS
LIN {X 91.015,Y -38.024,Z -101.602,A -90.000,B 90.000,C 0.000} C_DIS
LIN {X 90.639,Y -38.082,Z -102.269,A -90.000,B 90.000,C 0.000} C_DIS
LIN {X 90.473,Y -38.089,Z -102.595,A -90.000,B 90.000,C 0.000} C_DIS
LIN {X 90.261,Y -38.124,Z -103.054,A -90.000,B 90.000,C 0.000} C_DIS
LIN {X 90.095,Y -38.125,Z -103.461,A -90.000,B 90.000,C 0.000} C_DIS
LIN {X 90.030,Y -38.141,Z -103.648,A -90.000,B 90.000,C 0.000} C_DIS
LIN {X 89.963,Y -38.139,Z -103.948,A -90.000,B 90.000,C 0.000} C_DIS
LIN {X 89.956,Y -38.119,Z -104.102,A -90.000,B 90.000,C 0.000} C_DIS
LIN {X 89.958,Y -38.118,Z -104.173,A -90.000,B 90.000,C 0.000} C_DIS
LIN {X 90.011,Y -38.084,Z -104.566,A -90.000,B 90.000,C 0.000} C_DIS
LIN {X 90.205,Y -38.074,Z -105.581,A -90.000,B 90.000,C 0.000} C_DIS
LIN {X 90.351,Y -38.075,Z -106.324,A -90.000,B 90.000,C 0.000} C_DIS
LIN {X 90.382,Y -38.081,Z -106.521,A -90.000,B 90.000,C 0.000} C_DIS
LIN {X 90.412,Y -38.094,Z -106.777,A -90.000,B 90.000,C 0.000} C_DIS
LIN {X 90.513,Y -38.112,Z -107.883,A -90.000,B 90.000,C 0.000} C_DIS
LIN {X 90.549,Y -38.113,Z -108.383,A -90.000,B 90.000,C 0.000} C_DIS
LIN {X 90.554,Y -38.117,Z -108.554,A -90.000,B 90.000,C 0.000} C_DIS
LIN {X 90.554,Y -38.119,Z -108.593,A -90.000,B 90.000,C 0.000} C_DIS
LIN {X 90.545,Y -38.119,Z -108.793,A -90.000,B 90.000,C 0.000} C_DIS
LIN {X 90.514,Y -38.121,Z -109.211,A -90.000,B 90.000,C 0.000} C_DIS
LIN {X 90.436,Y -38.151,Z -110.490,A -90.000,B 90.000,C 0.000} C_DIS
LIN {X 90.425,Y -38.154,Z -110.656,A -90.000,B 90.000,C 0.000} C_DIS
LIN {X 90.389,Y -38.149,Z -110.985,A -90.000,B 90.000,C 0.000} C_DIS
LIN {X 90.325,Y -38.151,Z -111.461,A -90.000,B 90.000,C 0.000} C_DIS
LIN {X 90.280,Y -38.159,Z -111.825,A -90.000,B 90.000,C 0.000} C_DIS
LIN {X 90.145,Y -38.193,Z -112.761,A -90.000,B 90.000,C 0.000} C_DIS
LIN {X 89.990,Y -38.208,Z -113.716,A -90.000,B 90.000,C 0.000} C_DIS
LIN {X 89.859,Y -38.235,Z -114.555,A -90.000,B 90.000,C 0.000} C_DIS
LIN {X 89.673,Y -38.283,Z -115.593,A -90.000,B 90.000,C 0.000} C_DIS
LIN {X 89.653,Y -38.287,Z -115.722,A -90.000,B 90.000,C 0.000} C_DIS
LIN {X 89.563,Y -38.303,Z -116.327,A -90.000,B 90.000,C 0.000} C_DIS
LIN {X 89.448,Y -38.332,Z -117.135,A -90.000,B 90.000,C 0.000} C_DIS
LIN {X 89.393,Y -38.360,Z -117.571,A -90.000,B 90.000,C 0.000} C_DIS
LIN {X 89.341,Y -38.377,Z -118.883,A -90.000,B 90.000,C 0.000} C_DIS
LIN {X 89.330,Y -38.380,Z -119.339,A -90.000,B 90.000,C 0.000} C_DIS
LIN {X 89.329,Y -38.381,Z -119.373,A -90.000,B 90.000,C 0.000} C_DIS
LIN {X 89.341,Y -38.377,Z -119.784,A -90.000,B 90.000,C 0.000} C_DIS
LIN {X 89.373,Y -38.381,Z -120.673,A -90.000,B 90.000,C 0.000} C_DIS
LIN {X 89.420,Y -38.368,Z -121.333,A -90.000,B 90.000,C 0.000} C_DIS
LIN {X 89.448,Y -38.359,Z -121.847,A -90.000,B 90.000,C 0.000} C_DIS
LIN {X 89.484,Y -38.358,Z -122.409,A -90.000,B 90.000,C 0.000} C_DIS
LIN {X 89.536,Y -38.343,Z -122.855,A -90.000,B 90.000,C 0.000} C_DIS
LIN {X 89.545,Y -38.341,Z -122.953,A -90.000,B 90.000,C 0.000} C_DIS
LIN {X 89.572,Y -38.338,Z -123.327,A -90.000,B 90.000,C 0.000} C_DIS
LIN {X 89.584,Y -38.331,Z -123.737,A -90.000,B 90.000,C 0.000} C_DIS
LIN {X 89.616,Y -38.330,Z -124.521,A -90.000,B 90.000,C 0.000} C_DIS
LIN {X 89.649,Y -38.318,Z -124.879,A -90.000,B 90.000,C 0.000} C_DIS
LIN {X 89.670,Y -38.312,Z -125.198,A -90.000,B 90.000,C 0.000} C_DIS
LIN {X 89.675,Y -38.311,Z -125.302,A -90.000,B 90.000,C 0.000} C_DIS
LIN {X 89.678,Y -38.299,Z -125.846,A -90.000,B 90.000,C 0.000} C_DIS
LIN {X 89.659,Y -38.300,Z -126.427,A -90.000,B 90.000,C 0.000} C_DIS
LIN {X 89.638,Y -38.302,Z -127.060,A -90.000,B 90.000,C 0.000} C_DIS
LIN {X 89.623,Y -38.300,Z -127.451,A -90.000,B 90.000,C 0.000} C_DIS
LIN {X 89.595,Y -38.293,Z -127.958,A -90.000,B 90.000,C 0.000} C_DIS
LIN {X 89.568,Y -38.293,Z -128.327,A -90.000,B 90.000,C 0.000} C_DIS
LIN {X 89.476,Y -38.297,Z -129.463,A -90.000,B 90.000,C 0.000} C_DIS
LIN {X 89.394,Y -38.286,Z -130.485,A -90.000,B 90.000,C 0.000} C_DIS
LIN {X 89.272,Y -38.289,Z -131.727,A -90.000,B 90.000,C 0.000} C_DIS
LIN {X 89.181,Y -38.278,Z -132.876,A -90.000,B 90.000,C 0.000} C_DIS
LIN {X 89.048,Y -38.279,Z -134.303,A -90.000,B 90.000,C 0.000} C_DIS
LIN {X 88.930,Y -38.276,Z -135.887,A -90.000,B 90.000,C 0.000} C_DIS
LIN {X 88.843,Y -38.261,Z -137.293,A -90.000,B 90.000,C 0.000} C_DIS
LIN {X 88.701,Y -38.253,Z -139.274,A -90.000,B 90.000,C 0.000} C_DIS
LIN {X 88.612,Y -38.237,Z -140.732,A -90.000,B 90.000,C 0.000} C_DIS
LIN {X 88.425,Y -38.226,Z -143.063,A -90.000,B 90.000,C 0.000} C_DIS
LIN {X 88.326,Y -38.211,Z -144.437,A -90.000,B 90.000,C 0.000} C_DIS
LIN {X 88.317,Y -38.212,Z -144.544,A -90.000,B 90.000,C 0.000} C_DIS
LIN {X 88.256,Y -38.206,Z -145.146,A -90.000,B 90.000,C 0.000} C_DIS
LIN {X 88.063,Y -38.197,Z -147.098,A -90.000,B 90.000,C 0.000} C_DIS
LIN {X 87.948,Y -38.184,Z -148.346,A -90.000,B 90.000,C 0.000} C_DIS
LIN {X 87.910,Y -38.179,Z -148.688,A -90.000,B 90.000,C 0.000} C_DIS
LIN {X 87.802,Y -38.169,Z -149.587,A -90.000,B 90.000,C 0.000} C_DIS
LIN {X 87.606,Y -38.163,Z -151.116,A -90.000,B 90.000,C 0.000} C_DIS
LIN {X 87.441,Y -38.150,Z -152.362,A -90.000,B 90.000,C 0.000} C_DIS
LIN {X 87.423,Y -38.149,Z -152.496,A -90.000,B 90.000,C 0.000} C_DIS
LIN {X 87.315,Y -38.142,Z -153.195,A -90.000,B 90.000,C 0.000} C_DIS
LIN {X 87.022,Y -38.135,Z -155.025,A -90.000,B 90.000,C 0.000} C_DIS
LIN {X 86.851,Y -38.126,Z -156.070,A -90.000,B 90.000,C 0.000} C_DIS
LIN {X 86.817,Y -38.124,Z -156.271,A -90.000,B 90.000,C 0.000} C_DIS
LIN {X 86.716,Y -38.120,Z -156.805,A -90.000,B 90.000,C 0.000} C_DIS
LIN {X 86.370,Y -38.115,Z -158.571,A -90.000,B 90.000,C 0.000} C_DIS
LIN {X 86.104,Y -38.106,Z -159.901,A -90.000,B 90.000,C 0.000} C_DIS
LIN {X 86.076,Y -38.103,Z -160.033,A -90.000,B 90.000,C 0.000} C_DIS
LIN {X 85.985,Y -38.102,Z -160.427,A -90.000,B 90.000,C 0.000} C_DIS
LIN {X 85.583,Y -38.100,Z -162.137,A -90.000,B 90.000,C 0.000} C_DIS
LIN {X 85.255,Y -38.094,Z -163.515,A -90.000,B 90.000,C 0.000} C_DIS
LIN {X 85.113,Y -38.085,Z -164.070,A -90.000,B 90.000,C 0.000} C_DIS
LIN {X 84.160,Y -38.091,Z -167.485,A -90.000,B 90.000,C 0.000} C_DIS
LIN {X 84.115,Y -38.089,Z -167.639,A -90.000,B 90.000,C 0.000} C_DIS
LIN {X 83.109,Y -38.102,Z -170.912,A -90.000,B 90.000,C 0.000} C_DIS
LIN {X 82.974,Y -38.102,Z -171.335,A -90.000,B 90.000,C 0.000} C_DIS
LIN {X 82.010,Y -38.113,Z -174.351,A -90.000,B 90.000,C 0.000} C_DIS
LIN {X 81.818,Y -38.112,Z -174.969,A -90.000,B 90.000,C 0.000} C_DIS
LIN {X 81.055,Y -38.117,Z -177.388,A -90.000,B 90.000,C 0.000} C_DIS
LIN {X 80.999,Y -38.115,Z -177.578,A -90.000,B 90.000,C 0.000} C_DIS
LIN {X 80.441,Y -38.110,Z -179.504,A -90.000,B 90.000,C 0.000} C_DIS
LIN {X 80.238,Y -38.103,Z -180.228,A -90.000,B 90.000,C 0.000} C_DIS
LIN {X 80.143,Y -38.097,Z -180.568,A -90.000,B 90.000,C 0.000} C_DIS
LIN {X 79.763,Y -38.088,Z -181.969,A -90.000,B 90.000,C 0.000} C_DIS
LIN {X 79.496,Y -38.072,Z -182.993,A -90.000,B 90.000,C 0.000} C_DIS
LIN {X 79.361,Y -38.063,Z -183.487,A -90.000,B 90.000,C 0.000} C_DIS
LIN {X 79.027,Y -38.052,Z -184.758,A -90.000,B 90.000,C 0.000} C_DIS
LIN {X 78.856,Y -38.038,Z -185.438,A -90.000,B 90.000,C 0.000} C_DIS
LIN {X 78.807,Y -38.037,Z -185.627,A -90.000,B 90.000,C 0.000} C_DIS
LIN {X 78.621,Y -38.023,Z -186.307,A -90.000,B 90.000,C 0.000} C_DIS
LIN {X 78.303,Y -38.011,Z -187.509,A -90.000,B 90.000,C 0.000} C_DIS
LIN {X 78.183,Y -38.002,Z -187.986,A -90.000,B 90.000,C 0.000} C_DIS
LIN {X 78.136,Y -38.001,Z -188.159,A -90.000,B 90.000,C 0.000} C_DIS
LIN {X 77.892,Y -37.985,Z -189.016,A -90.000,B 90.000,C 0.000} C_DIS
LIN {X 77.818,Y -37.983,Z -189.286,A -90.000,B 90.000,C 0.000} C_DIS
LIN {X 77.575,Y -37.975,Z -190.168,A -90.000,B 90.000,C 0.000} C_DIS
LIN {X 77.493,Y -37.970,Z -190.474,A -90.000,B 90.000,C 0.000} C_DIS
LIN {X 77.451,Y -37.970,Z -190.621,A -90.000,B 90.000,C 0.000} C_DIS
LIN {X 77.126,Y -37.955,Z -191.686,A -90.000,B 90.000,C 0.000} C_DIS
LIN {X 76.759,Y -37.946,Z -192.921,A -90.000,B 90.000,C 0.000} C_DIS
LIN {X 76.681,Y -37.943,Z -193.188,A -90.000,B 90.000,C 0.000} C_DIS
LIN {X 76.604,Y -37.937,Z -193.431,A -90.000,B 90.000,C 0.000} C_DIS
LIN {X 76.242,Y -37.926,Z -194.531,A -90.000,B 90.000,C 0.000} C_DIS
LIN {X 75.755,Y -37.918,Z -196.032,A -90.000,B 90.000,C 0.000} C_DIS
LIN {X 75.664,Y -37.913,Z -196.300,A -90.000,B 90.000,C 0.000} C_DIS
LIN {X 75.152,Y -37.904,Z -197.740,A -90.000,B 90.000,C 0.000} C_DIS
LIN {X 74.580,Y -37.899,Z -199.364,A -90.000,B 90.000,C 0.000} C_DIS
LIN {X 74.491,Y -37.896,Z -199.610,A -90.000,B 90.000,C 0.000} C_DIS
LIN {X 73.935,Y -37.891,Z -201.089,A -90.000,B 90.000,C 0.000} C_DIS
LIN {X 73.017,Y -37.886,Z -203.537,A -90.000,B 90.000,C 0.000} C_DIS
LIN {X 71.276,Y -37.878,Z -207.962,A -90.000,B 90.000,C 0.000} C_DIS
LIN {X 69.332,Y -37.872,Z -212.693,A -90.000,B 90.000,C 0.000} C_DIS
LIN {X 69.170,Y -37.868,Z -213.079,A -90.000,B 90.000,C 0.000} C_DIS
LIN {X 67.369,Y -37.863,Z -217.282,A -90.000,B 90.000,C 0.000} C_DIS
LIN {X 67.169,Y -37.863,Z -217.746,A -90.000,B 90.000,C 0.000} C_DIS
LIN {X 66.972,Y -37.859,Z -218.193,A -90.000,B 90.000,C 0.000} C_DIS
LIN {X 64.813,Y -37.858,Z -222.993,A -90.000,B 90.000,C 0.000} C_DIS
LIN {X 64.642,Y -37.855,Z -223.363,A -90.000,B 90.000,C 0.000} C_DIS
LIN {X 63.687,Y -37.855,Z -225.369,A -90.000,B 90.000,C 0.000} C_DIS
LIN {X 62.225,Y -37.862,Z -228.458,A -90.000,B 90.000,C 0.000} C_DIS
LIN {X 62.100,Y -37.860,Z -228.717,A -90.000,B 90.000,C 0.000} C_DIS
LIN {X 61.974,Y -37.859,Z -228.967,A -90.000,B 90.000,C 0.000} C_DIS
LIN {X 61.268,Y -37.858,Z -230.355,A -90.000,B 90.000,C 0.000} C_DIS
LIN {X 59.643,Y -37.882,Z -233.599,A -90.000,B 90.000,C 0.000} C_DIS
LIN {X 59.543,Y -37.882,Z -233.796,A -90.000,B 90.000,C 0.000} C_DIS
LIN {X 59.413,Y -37.876,Z -234.047,A -90.000,B 90.000,C 0.000} C_DIS
LIN {X 59.307,Y -37.875,Z -234.244,A -90.000,B 90.000,C 0.000} C_DIS
LIN {X 58.707,Y -37.875,Z -235.335,A -90.000,B 90.000,C 0.000} C_DIS
LIN {X 56.777,Y -37.927,Z -238.953,A -90.000,B 90.000,C 0.000} C_DIS
LIN {X 56.678,Y -37.927,Z -239.145,A -90.000,B 90.000,C 0.000} C_DIS
LIN {X 56.490,Y -37.923,Z -239.498,A -90.000,B 90.000,C 0.000} C_DIS
LIN {X 56.167,Y -37.923,Z -240.093,A -90.000,B 90.000,C 0.000} C_DIS
LIN {X 55.973,Y -37.926,Z -240.441,A -90.000,B 90.000,C 0.000} C_DIS
LIN {X 54.504,Y -37.990,Z -243.004,A -90.000,B 90.000,C 0.000} C_DIS
LIN {X 54.344,Y -37.994,Z -243.277,A -90.000,B 90.000,C 0.000} C_DIS
LIN {X 54.174,Y -37.994,Z -243.561,A -90.000,B 90.000,C 0.000} C_DIS
LIN {X 54.174,Y -60.000,Z -243.561,A -90.000,B 90.000,C 0.000} C_DIS
LIN {X -85.807,Y -60.000,Z -243.561,A -90.000,B 90.000,C 0.000} C_DIS
LIN {X -85.807,Y -38.597,Z -243.561,A -90.000,B 90.000,C 0.000} C_DIS
LIN {X -85.635,Y -38.370,Z -243.074,A -90.000,B 90.000,C 0.000} C_DIS
LIN {X -85.562,Y -38.319,Z -242.943,A -90.000,B 90.000,C 0.000} C_DIS
LIN {X -85.288,Y -38.206,Z -242.580,A -90.000,B 90.000,C 0.000} C_DIS
LIN {X -84.809,Y -38.154,Z -242.180,A -90.000,B 90.000,C 0.000} C_DIS
LIN {X -83.869,Y -38.165,Z -241.578,A -90.000,B 90.000,C 0.000} C_DIS
LIN {X -83.607,Y -38.165,Z -241.413,A -90.000,B 90.000,C 0.000} C_DIS
LIN {X -82.923,Y -38.159,Z -240.987,A -90.000,B 90.000,C 0.000} C_DIS
LIN {X -80.520,Y -38.159,Z -239.534,A -90.000,B 90.000,C 0.000} C_DIS
LIN {X -77.306,Y -38.187,Z -237.639,A -90.000,B 90.000,C 0.000} C_DIS
LIN {X -75.605,Y -38.187,Z -236.647,A -90.000,B 90.000,C 0.000} C_DIS
LIN {X -74.690,Y -38.178,Z -236.122,A -90.000,B 90.000,C 0.000} C_DIS
LIN {X -73.665,Y -38.180,Z -235.555,A -90.000,B 90.000,C 0.000} C_DIS
LIN {X -70.718,Y -38.195,Z -233.940,A -90.000,B 90.000,C 0.000} C_DIS
LIN {X -67.423,Y -38.197,Z -232.149,A -90.000,B 90.000,C 0.000} C_DIS
LIN {X -67.033,Y -38.198,Z -231.941,A -90.000,B 90.000,C 0.000} C_DIS
LIN {X -66.118,Y -38.192,Z -231.460,A -90.000,B 90.000,C 0.000} C_DIS
LIN {X -64.431,Y -38.197,Z -230.598,A -90.000,B 90.000,C 0.000} C_DIS
LIN {X -58.401,Y -38.211,Z -227.516,A -90.000,B 90.000,C 0.000} C_DIS
LIN {X -57.505,Y -38.207,Z -227.062,A -90.000,B 90.000,C 0.000} C_DIS
LIN {X -56.763,Y -38.207,Z -226.694,A -90.000,B 90.000,C 0.000} C_DIS
LIN {X -49.353,Y -38.202,Z -223.026,A -90.000,B 90.000,C 0.000} C_DIS
LIN {X -45.889,Y -38.209,Z -221.329,A -90.000,B 90.000,C 0.000} C_DIS
LIN {X -43.808,Y -38.210,Z -220.312,A -90.000,B 90.000,C 0.000} C_DIS
LIN {X -42.205,Y -38.213,Z -219.533,A -90.000,B 90.000,C 0.000} C_DIS
LIN {X -41.307,Y -38.219,Z -219.094,A -90.000,B 90.000,C 0.000} C_DIS
LIN {X -37.796,Y -38.232,Z -217.353,A -90.000,B 90.000,C 0.000} C_DIS
LIN {X -35.356,Y -38.233,Z -216.149,A -90.000,B 90.000,C 0.000} C_DIS
LIN {X -34.302,Y -38.240,Z -215.624,A -90.000,B 90.000,C 0.000} C_DIS
LIN {X -33.865,Y -38.240,Z -215.401,A -90.000,B 90.000,C 0.000} C_DIS
LIN {X -32.735,Y -38.237,Z -214.815,A -90.000,B 90.000,C 0.000} C_DIS
LIN {X -31.532,Y -38.244,Z -214.212,A -90.000,B 90.000,C 0.000} C_DIS
LIN {X -30.648,Y -38.252,Z -213.766,A -90.000,B 90.000,C 0.000} C_DIS
LIN {X -29.395,Y -38.263,Z -213.134,A -90.000,B 90.000,C 0.000} C_DIS
LIN {X -28.311,Y -38.282,Z -212.577,A -90.000,B 90.000,C 0.000} C_DIS
LIN {X -27.864,Y -38.284,Z -212.337,A -90.000,B 90.000,C 0.000} C_DIS
LIN {X -26.042,Y -38.303,Z -211.352,A -90.000,B 90.000,C 0.000} C_DIS
LIN {X -24.439,Y -38.310,Z -210.467,A -90.000,B 90.000,C 0.000} C_DIS
LIN {X -24.178,Y -38.315,Z -210.321,A -90.000,B 90.000,C 0.000} C_DIS
LIN {X -23.520,Y -38.331,Z -209.950,A -90.000,B 90.000,C 0.000} C_DIS
LIN {X -22.477,Y -38.332,Z -209.340,A -90.000,B 90.000,C 0.000} C_DIS
LIN {X -20.750,Y -38.319,Z -208.304,A -90.000,B 90.000,C 0.000} C_DIS
LIN {X -19.971,Y -38.319,Z -207.833,A -90.000,B 90.000,C 0.000} C_DIS
LIN {X -19.099,Y -38.332,Z -207.297,A -90.000,B 90.000,C 0.000} C_DIS
LIN {X -17.465,Y -38.328,Z -206.232,A -90.000,B 90.000,C 0.000} C_DIS
LIN {X -16.546,Y -38.332,Z -205.629,A -90.000,B 90.000,C 0.000} C_DIS
LIN {X -15.905,Y -38.339,Z -205.219,A -90.000,B 90.000,C 0.000} C_DIS
LIN {X -15.570,Y -38.348,Z -205.001,A -90.000,B 90.000,C 0.000} C_DIS
LIN {X -15.355,Y -38.353,Z -204.857,A -90.000,B 90.000,C 0.000} C_DIS
LIN {X -14.907,Y -38.356,Z -204.544,A -90.000,B 90.000,C 0.000} C_DIS
LIN {X -12.178,Y -38.375,Z -202.643,A -90.000,B 90.000,C 0.000} C_DIS
LIN {X -11.491,Y -38.392,Z -202.156,A -90.000,B 90.000,C 0.000} C_DIS
LIN {X -10.571,Y -38.398,Z -201.464,A -90.000,B 90.000,C 0.000} C_DIS
LIN {X -8.541,Y -38.410,Z -199.937,A -90.000,B 90.000,C 0.000} C_DIS
LIN {X -7.771,Y -38.427,Z -199.350,A -90.000,B 90.000,C 0.000} C_DIS
LIN {X -5.517,Y -38.433,Z -197.524,A -90.000,B 90.000,C 0.000} C_DIS
LIN {X -4.953,Y -38.435,Z -197.070,A -90.000,B 90.000,C 0.000} C_DIS
LIN {X -4.230,Y -38.449,Z -196.481,A -90.000,B 90.000,C 0.000} C_DIS
LIN {X -1.503,Y -38.438,Z -194.104,A -90.000,B 90.000,C 0.000} C_DIS
LIN {X -0.756,Y -38.449,Z -193.459,A -90.000,B 90.000,C 0.000} C_DIS
LIN {X -0.170,Y -38.450,Z -192.937,A -90.000,B 90.000,C 0.000} C_DIS
LIN {X 1.967,Y -38.415,Z -190.934,A -90.000,B 90.000,C 0.000} C_DIS
LIN {X 2.848,Y -38.409,Z -190.103,A -90.000,B 90.000,C 0.000} C_DIS
LIN {X 3.128,Y -38.409,Z -189.845,A -90.000,B 90.000,C 0.000} C_DIS
LIN {X 5.353,Y -38.365,Z -187.673,A -90.000,B 90.000,C 0.000} C_DIS
LIN {X 5.661,Y -38.365,Z -187.368,A -90.000,B 90.000,C 0.000} C_DIS
LIN {X 6.340,Y -38.355,Z -186.703,A -90.000,B 90.000,C 0.000} C_DIS
LIN {X 8.137,Y -38.321,Z -184.922,A -90.000,B 90.000,C 0.000} C_DIS
LIN {X 9.136,Y -38.320,Z -183.916,A -90.000,B 90.000,C 0.000} C_DIS
LIN {X 9.621,Y -38.313,Z -183.434,A -90.000,B 90.000,C 0.000} C_DIS
LIN {X 11.207,Y -38.291,Z -181.873,A -90.000,B 90.000,C 0.000} C_DIS
LIN {X 12.180,Y -38.291,Z -180.905,A -90.000,B 90.000,C 0.000} C_DIS
LIN {X 12.649,Y -38.277,Z -180.421,A -90.000,B 90.000,C 0.000} C_DIS
LIN {X 13.597,Y -38.267,Z -179.499,A -90.000,B 90.000,C 0.000} C_DIS
LIN {X 14.648,Y -38.263,Z -178.500,A -90.000,B 90.000,C 0.000} C_DIS
LIN {X 15.548,Y -38.258,Z -177.646,A -90.000,B 90.000,C 0.000} C_DIS
LIN {X 16.078,Y -38.259,Z -177.148,A -90.000,B 90.000,C 0.000} C_DIS
LIN {X 17.997,Y -38.270,Z -175.349,A -90.000,B 90.000,C 0.000} C_DIS
LIN {X 18.626,Y -38.282,Z -174.753,A -90.000,B 90.000,C 0.000} C_DIS
LIN {X 19.097,Y -38.289,Z -174.303,A -90.000,B 90.000,C 0.000} C_DIS
LIN {X 19.890,Y -38.304,Z -173.541,A -90.000,B 90.000,C 0.000} C_DIS
LIN {X 20.462,Y -38.320,Z -172.970,A -90.000,B 90.000,C 0.000} C_DIS
LIN {X 20.994,Y -38.330,Z -172.426,A -90.000,B 90.000,C 0.000} C_DIS
LIN {X 21.420,Y -38.345,Z -171.987,A -90.000,B 90.000,C 0.000} C_DIS
LIN {X 21.956,Y -38.362,Z -171.388,A -90.000,B 90.000,C 0.000} C_DIS
LIN {X 22.353,Y -38.373,Z -170.941,A -90.000,B 90.000,C 0.000} C_DIS
LIN {X 22.934,Y -38.389,Z -170.274,A -90.000,B 90.000,C 0.000} C_DIS
LIN {X 23.034,Y -38.394,Z -170.158,A -90.000,B 90.000,C 0.000} C_DIS
LIN {X 23.293,Y -38.402,Z -169.837,A -90.000,B 90.000,C 0.000} C_DIS
LIN {X 24.375,Y -38.426,Z -168.470,A -90.000,B 90.000,C 0.000} C_DIS
LIN {X 24.512,Y -38.427,Z -168.289,A -90.000,B 90.000,C 0.000} C_DIS
LIN {X 24.859,Y -38.437,Z -167.823,A -90.000,B 90.000,C 0.000} C_DIS
LIN {X 25.839,Y -38.458,Z -166.485,A -90.000,B 90.000,C 0.000} C_DIS
LIN {X 25.978,Y -38.458,Z -166.290,A -90.000,B 90.000,C 0.000} C_DIS
LIN {X 26.358,Y -38.467,Z -165.747,A -90.000,B 90.000,C 0.000} C_DIS
LIN {X 26.819,Y -38.476,Z -165.083,A -90.000,B 90.000,C 0.000} C_DIS
LIN {X 27.017,Y -38.489,Z -164.791,A -90.000,B 90.000,C 0.000} C_DIS
LIN {X 27.278,Y -38.497,Z -164.413,A -90.000,B 90.000,C 0.000} C_DIS
LIN {X 28.162,Y -38.516,Z -163.100,A -90.000,B 90.000,C 0.000} C_DIS
LIN {X 28.542,Y -38.538,Z -162.527,A -90.000,B 90.000,C 0.000} C_DIS
LIN {X 28.715,Y -38.545,Z -162.268,A -90.000,B 90.000,C 0.000} C_DIS
LIN {X 29.403,Y -38.565,Z -161.189,A -90.000,B 90.000,C 0.000} C_DIS
LIN {X 29.930,Y -38.596,Z -160.350,A -90.000,B 90.000,C 0.000} C_DIS
LIN {X 30.022,Y -38.600,Z -160.188,A -90.000,B 90.000,C 0.000} C_DIS
LIN {X 30.211,Y -38.610,Z -159.858,A -90.000,B 90.000,C 0.000} C_DIS
LIN {X 30.724,Y -38.669,Z -158.950,A -90.000,B 90.000,C 0.000} C_DIS
LIN {X 30.957,Y -38.702,Z -158.536,A -90.000,B 90.000,C 0.000} C_DIS
LIN {X 31.057,Y -38.716,Z -158.333,A -90.000,B 90.000,C 0.000} C_DIS
LIN {X 31.338,Y -38.755,Z -157.778,A -90.000,B 90.000,C 0.000} C_DIS
LIN {X 31.428,Y -38.768,Z -157.576,A -90.000,B 90.000,C 0.000} C_DIS
LIN {X 31.737,Y -38.853,Z -156.871,A -90.000,B 90.000,C 0.000} C_DIS
LIN {X 31.923,Y -38.917,Z -156.322,A -90.000,B 90.000,C 0.000} C_DIS
LIN {X 31.999,Y -38.941,Z -156.119,A -90.000,B 90.000,C 0.000} C_DIS
LIN {X 32.092,Y -38.993,Z -155.638,A -90.000,B 90.000,C 0.000} C_DIS
LIN {X 32.141,Y -39.026,Z -155.398,A -90.000,B 90.000,C 0.000} C_DIS
LIN {X 31.610,Y -39.013,Z -155.450,A -90.000,B 90.000,C 0.000} C_DIS
LIN {X 31.532,Y -39.013,Z -155.458,A -90.000,B 90.000,C 0.000} C_DIS
LIN {X 30.930,Y -39.000,Z -155.613,A -90.000,B 90.000,C 0.000} C_DIS
LIN {X 30.808,Y -38.999,Z -155.636,A -90.000,B 90.000,C 0.000} C_DIS
LIN {X 30.623,Y -38.997,Z -155.666,A -90.000,B 90.000,C 0.000} C_DIS
LIN {X 30.422,Y -38.997,Z -155.689,A -90.000,B 90.000,C 0.000} C_DIS
LIN {X 30.351,Y -38.998,Z -155.692,A -90.000,B 90.000,C 0.000} C_DIS
LIN {X 30.087,Y -39.008,Z -155.695,A -90.000,B 90.000,C 0.000} C_DIS
LIN {X 29.819,Y -39.014,Z -155.696,A -90.000,B 90.000,C 0.000} C_DIS
LIN {X 28.857,Y -39.010,Z -155.820,A -90.000,B 90.000,C 0.000} C_DIS
LIN {X 28.548,Y -39.005,Z -155.858,A -90.000,B 90.000,C 0.000} C_DIS
LIN {X 28.432,Y -39.005,Z -155.864,A -90.000,B 90.000,C 0.000} C_DIS
LIN {X 28.285,Y -39.006,Z -155.863,A -90.000,B 90.000,C 0.000} C_DIS
LIN {X 28.149,Y -39.005,Z -155.852,A -90.000,B 90.000,C 0.000} C_DIS
LIN {X 27.894,Y -39.006,Z -155.823,A -90.000,B 90.000,C 0.000} C_DIS
LIN {X 27.762,Y -39.007,Z -155.803,A -90.000,B 90.000,C 0.000} C_DIS
LIN {X 27.605,Y -39.009,Z -155.771,A -90.000,B 90.000,C 0.000} C_DIS
LIN {X 27.499,Y -39.012,Z -155.741,A -90.000,B 90.000,C 0.000} C_DIS
LIN {X 27.406,Y -39.015,Z -155.710,A -90.000,B 90.000,C 0.000} C_DIS
LIN {X 27.280,Y -39.019,Z -155.659,A -90.000,B 90.000,C 0.000} C_DIS
LIN {X 27.099,Y -39.025,Z -155.583,A -90.000,B 90.000,C 0.000} C_DIS
LIN {X 26.695,Y -39.049,Z -155.339,A -90.000,B 90.000,C 0.000} C_DIS
LIN {X 26.560,Y -39.056,Z -155.234,A -90.000,B 90.000,C 0.000} C_DIS
LIN {X 26.500,Y -39.056,Z -155.184,A -90.000,B 90.000,C 0.000} C_DIS
LIN {X 26.421,Y -39.057,Z -155.114,A -90.000,B 90.000,C 0.000} C_DIS
LIN {X 26.370,Y -39.056,Z -155.063,A -90.000,B 90.000,C 0.000} C_DIS
LIN {X 26.294,Y -39.054,Z -154.981,A -90.000,B 90.000,C 0.000} C_DIS
LIN {X 26.194,Y -39.052,Z -154.857,A -90.000,B 90.000,C 0.000} C_DIS
LIN {X 25.865,Y -39.046,Z -154.444,A -90.000,B 90.000,C 0.000} C_DIS
LIN {X 25.462,Y -39.045,Z -153.941,A -90.000,B 90.000,C 0.000} C_DIS
LIN {X 25.389,Y -39.041,Z -153.849,A -90.000,B 90.000,C 0.000} C_DIS
LIN {X 25.327,Y -39.037,Z -153.765,A -90.000,B 90.000,C 0.000} C_DIS
LIN {X 25.228,Y -39.021,Z -153.621,A -90.000,B 90.000,C 0.000} C_DIS
LIN {X 25.165,Y -39.009,Z -153.523,A -90.000,B 90.000,C 0.000} C_DIS
LIN {X 25.119,Y -39.001,Z -153.443,A -90.000,B 90.000,C 0.000} C_DIS
LIN {X 24.987,Y -38.978,Z -153.142,A -90.000,B 90.000,C 0.000} C_DIS
LIN {X 24.924,Y -38.967,Z -152.963,A -90.000,B 90.000,C 0.000} C_DIS
LIN {X 24.884,Y -38.960,Z -152.828,A -90.000,B 90.000,C 0.000} C_DIS
LIN {X 24.858,Y -38.955,Z -152.718,A -90.000,B 90.000,C 0.000} C_DIS
LIN {X 24.820,Y -38.949,Z -152.437,A -90.000,B 90.000,C 0.000} C_DIS
LIN {X 24.809,Y -38.947,Z -152.258,A -90.000,B 90.000,C 0.000} C_DIS
LIN {X 24.805,Y -38.946,Z -152.129,A -90.000,B 90.000,C 0.000} C_DIS
LIN {X 24.805,Y -38.945,Z -151.954,A -90.000,B 90.000,C 0.000} C_DIS
LIN {X 24.815,Y -38.947,Z -151.805,A -90.000,B 90.000,C 0.000} C_DIS
LIN {X 24.842,Y -38.949,Z -151.624,A -90.000,B 90.000,C 0.000} C_DIS
LIN {X 24.859,Y -38.951,Z -151.546,A -90.000,B 90.000,C 0.000} C_DIS
LIN {X 24.997,Y -38.943,Z -150.931,A -90.000,B 90.000,C 0.000} C_DIS
LIN {X 25.184,Y -38.917,Z -150.119,A -90.000,B 90.000,C 0.000} C_DIS
LIN {X 25.214,Y -38.908,Z -149.992,A -90.000,B 90.000,C 0.000} C_DIS
LIN {X 25.411,Y -38.859,Z -149.227,A -90.000,B 90.000,C 0.000} C_DIS
LIN {X 25.455,Y -38.851,Z -149.088,A -90.000,B 90.000,C 0.000} C_DIS
LIN {X 25.482,Y -38.847,Z -149.018,A -90.000,B 90.000,C 0.000} C_DIS
LIN {X 25.880,Y -38.791,Z -148.056,A -90.000,B 90.000,C 0.000} C_DIS
LIN {X 25.912,Y -38.784,Z -147.984,A -90.000,B 90.000,C 0.000} C_DIS
LIN {X 25.983,Y -38.775,Z -147.842,A -90.000,B 90.000,C 0.000} C_DIS
LIN {X 26.158,Y -38.759,Z -147.526,A -90.000,B 90.000,C 0.000} C_DIS
LIN {X 26.319,Y -38.747,Z -147.247,A -90.000,B 90.000,C 0.000} C_DIS
LIN {X 26.495,Y -38.728,Z -146.959,A -90.000,B 90.000,C 0.000} C_DIS
LIN {X 26.661,Y -38.720,Z -146.724,A -90.000,B 90.000,C 0.000} C_DIS
LIN {X 26.904,Y -38.720,Z -146.425,A -90.000,B 90.000,C 0.000} C_DIS
LIN {X 26.979,Y -38.717,Z -146.334,A -90.000,B 90.000,C 0.000} C_DIS
LIN {X 27.505,Y -38.696,Z -145.697,A -90.000,B 90.000,C 0.000} C_DIS
LIN {X 26.909,Y -38.600,Z -145.978,A -90.000,B 90.000,C 0.000} C_DIS
LIN {X 26.650,Y -38.557,Z -146.098,A -90.000,B 90.000,C 0.000} C_DIS
LIN {X 26.166,Y -38.459,Z -146.309,A -90.000,B 90.000,C 0.000} C_DIS
LIN {X 25.382,Y -38.293,Z -146.630,A -90.000,B 90.000,C 0.000} C_DIS
LIN {X 25.095,Y -38.230,Z -146.740,A -90.000,B 90.000,C 0.000} C_DIS
LIN {X 24.914,Y -38.190,Z -146.807,A -90.000,B 90.000,C 0.000} C_DIS
LIN {X 24.745,Y -38.148,Z -146.865,A -90.000,B 90.000,C 0.000} C_DIS
LIN {X 24.433,Y -38.056,Z -146.954,A -90.000,B 90.000,C 0.000} C_DIS
LIN {X 24.155,Y -37.970,Z -147.019,A -90.000,B 90.000,C 0.000} C_DIS
LIN {X 24.016,Y -37.922,Z -147.041,A -90.000,B 90.000,C 0.000} C_DIS
LIN {X 23.831,Y -37.870,Z -147.076,A -90.000,B 90.000,C 0.000} C_DIS
LIN {X 23.676,Y -37.821,Z -147.093,A -90.000,B 90.000,C 0.000} C_DIS
LIN {X 23.534,Y -37.774,Z -147.101,A -90.000,B 90.000,C 0.000} C_DIS
LIN {X 23.329,Y -37.700,Z -147.095,A -90.000,B 90.000,C 0.000} C_DIS
LIN {X 23.284,Y -37.683,Z -147.089,A -90.000,B 90.000,C 0.000} C_DIS
LIN {X 21.980,Y -37.688,Z -147.677,A -90.000,B 90.000,C 0.000} C_DIS
LIN {X 21.059,Y -37.705,Z -148.080,A -90.000,B 90.000,C 0.000} C_DIS
LIN {X 20.803,Y -37.705,Z -148.184,A -90.000,B 90.000,C 0.000} C_DIS
LIN {X 20.197,Y -37.697,Z -148.420,A -90.000,B 90.000,C 0.000} C_DIS
LIN {X 19.154,Y -37.686,Z -148.820,A -90.000,B 90.000,C 0.000} C_DIS
LIN {X 18.704,Y -37.692,Z -148.985,A -90.000,B 90.000,C 0.000} C_DIS
LIN {X 18.290,Y -37.704,Z -149.132,A -90.000,B 90.000,C 0.000} C_DIS
LIN {X 17.348,Y -37.724,Z -149.454,A -90.000,B 90.000,C 0.000} C_DIS
LIN {X 16.880,Y -37.732,Z -149.611,A -90.000,B 90.000,C 0.000} C_DIS
LIN {X 15.672,Y -37.742,Z -150.001,A -90.000,B 90.000,C 0.000} C_DIS
LIN {X 14.277,Y -37.751,Z -150.436,A -90.000,B 90.000,C 0.000} C_DIS
LIN {X 13.845,Y -37.747,Z -150.562,A -90.000,B 90.000,C 0.000} C_DIS
LIN {X 13.514,Y -37.744,Z -150.653,A -90.000,B 90.000,C 0.000} C_DIS
LIN {X 13.243,Y -37.742,Z -150.724,A -90.000,B 90.000,C 0.000} C_DIS
LIN {X 11.138,Y -37.777,Z -151.219,A -90.000,B 90.000,C 0.000} C_DIS
LIN {X 10.712,Y -37.780,Z -151.312,A -90.000,B 90.000,C 0.000} C_DIS
LIN {X 9.867,Y -37.775,Z -151.473,A -90.000,B 90.000,C 0.000} C_DIS
LIN {X 9.627,Y -37.772,Z -151.518,A -90.000,B 90.000,C 0.000} C_DIS
LIN {X 8.933,Y -37.764,Z -151.642,A -90.000,B 90.000,C 0.000} C_DIS
LIN {X 8.432,Y -37.769,Z -151.723,A -90.000,B 90.000,C 0.000} C_DIS
LIN {X 7.528,Y -37.798,Z -151.852,A -90.000,B 90.000,C 0.000} C_DIS
LIN {X 7.304,Y -37.798,Z -151.876,A -90.000,B 90.000,C 0.000} C_DIS
LIN {X 5.178,Y -37.764,Z -152.054,A -90.000,B 90.000,C 0.000} C_DIS
LIN {X 4.823,Y -37.764,Z -152.079,A -90.000,B 90.000,C 0.000} C_DIS
LIN {X 4.619,Y -37.765,Z -152.091,A -90.000,B 90.000,C 0.000} C_DIS
LIN {X 4.230,Y -37.780,Z -152.105,A -90.000,B 90.000,C 0.000} C_DIS
LIN {X 3.807,Y -37.781,Z -152.102,A -90.000,B 90.000,C 0.000} C_DIS
LIN {X 1.397,Y -37.741,Z -152.016,A -90.000,B 90.000,C 0.000} C_DIS
LIN {X 0.643,Y -37.740,Z -151.982,A -90.000,B 90.000,C 0.000} C_DIS
LIN {X 0.552,Y -37.742,Z -151.976,A -90.000,B 90.000,C 0.000} C_DIS
LIN {X 0.115,Y -37.749,Z -151.919,A -90.000,B 90.000,C 0.000} C_DIS
LIN {X -0.527,Y -37.740,Z -151.809,A -90.000,B 90.000,C 0.000} C_DIS
LIN {X -2.442,Y -37.720,Z -151.491,A -90.000,B 90.000,C 0.000} C_DIS
LIN {X -3.271,Y -37.717,Z -151.349,A -90.000,B 90.000,C 0.000} C_DIS
LIN {X -3.373,Y -37.715,Z -151.329,A -90.000,B 90.000,C 0.000} C_DIS
LIN {X -3.489,Y -37.713,Z -151.304,A -90.000,B 90.000,C 0.000} C_DIS
LIN {X -3.700,Y -37.712,Z -151.251,A -90.000,B 90.000,C 0.000} C_DIS
LIN {X -7.362,Y -37.697,Z -150.192,A -90.000,B 90.000,C 0.000} C_DIS
LIN {X -7.543,Y -37.689,Z -150.128,A -90.000,B 90.000,C 0.000} C_DIS
LIN {X -7.788,Y -37.684,Z -150.034,A -90.000,B 90.000,C 0.000} C_DIS
LIN {X -11.323,Y -37.690,Z -148.584,A -90.000,B 90.000,C 0.000} C_DIS
LIN {X -11.513,Y -37.684,Z -148.494,A -90.000,B 90.000,C 0.000} C_DIS
LIN {X -11.730,Y -37.674,Z -148.386,A -90.000,B 90.000,C 0.000} C_DIS
LIN {X -11.832,Y -37.672,Z -148.334,A -90.000,B 90.000,C 0.000} C_DIS
LIN {X -14.111,Y -37.695,Z -147.104,A -90.000,B 90.000,C 0.000} C_DIS
LIN {X -15.243,Y -37.704,Z -146.488,A -90.000,B 90.000,C 0.000} C_DIS
LIN {X -15.614,Y -37.691,Z -146.258,A -90.000,B 90.000,C 0.000} C_DIS
LIN {X -15.754,Y -37.685,Z -146.169,A -90.000,B 90.000,C 0.000} C_DIS
LIN {X -15.896,Y -37.683,Z -146.075,A -90.000,B 90.000,C 0.000} C_DIS
LIN {X -16.207,Y -37.686,Z -145.864,A -90.000,B 90.000,C 0.000} C_DIS
LIN {X -17.379,Y -37.700,Z -145.065,A -90.000,B 90.000,C 0.000} C_DIS
LIN {X -18.885,Y -37.721,Z -144.048,A -90.000,B 90.000,C 0.000} C_DIS
LIN {X -19.349,Y -37.726,Z -143.731,A -90.000,B 90.000,C 0.000} C_DIS
LIN {X -19.760,Y -37.717,Z -143.408,A -90.000,B 90.000,C 0.000} C_DIS
LIN {X -20.396,Y -37.726,Z -142.887,A -90.000,B 90.000,C 0.000} C_DIS
LIN {X -20.991,Y -37.745,Z -142.392,A -90.000,B 90.000,C 0.000} C_DIS
LIN {X -21.288,Y -37.753,Z -142.141,A -90.000,B 90.000,C 0.000} C_DIS
LIN {X -22.321,Y -37.772,Z -141.254,A -90.000,B 90.000,C 0.000} C_DIS
LIN {X -22.656,Y -37.784,Z -140.961,A -90.000,B 90.000,C 0.000} C_DIS
LIN {X -22.824,Y -37.787,Z -140.808,A -90.000,B 90.000,C 0.000} C_DIS
LIN {X -22.980,Y -37.785,Z -140.654,A -90.000,B 90.000,C 0.000} C_DIS
LIN {X -23.301,Y -37.788,Z -140.327,A -90.000,B 90.000,C 0.000} C_DIS
LIN {X -24.802,Y -37.855,Z -138.743,A -90.000,B 90.000,C 0.000} C_DIS
LIN {X -25.541,Y -37.896,Z -137.954,A -90.000,B 90.000,C 0.000} C_DIS
LIN {X -25.901,Y -37.914,Z -137.565,A -90.000,B 90.000,C 0.000} C_DIS
LIN {X -25.970,Y -37.913,Z -137.484,A -90.000,B 90.000,C 0.000} C_DIS
LIN {X -26.078,Y -37.912,Z -137.353,A -90.000,B 90.000,C 0.000} C_DIS
LIN {X -26.327,Y -37.922,Z -137.036,A -90.000,B 90.000,C 0.000} C_DIS
LIN {X -27.021,Y -37.959,Z -136.142,A -90.000,B 90.000,C 0.000} C_DIS
LIN {X -27.200,Y -37.964,Z -135.903,A -90.000,B 90.000,C 0.000} C_DIS
LIN {X -28.049,Y -37.993,Z -134.754,A -90.000,B 90.000,C 0.000} C_DIS
LIN {X -28.356,Y -37.999,Z -134.331,A -90.000,B 90.000,C 0.000} C_DIS
LIN {X -28.435,Y -38.001,Z -134.218,A -90.000,B 90.000,C 0.000} C_DIS
LIN {X -28.503,Y -38.000,Z -134.112,A -90.000,B 90.000,C 0.000} C_DIS
LIN {X -28.620,Y -37.998,Z -133.923,A -90.000,B 90.000,C 0.000} C_DIS
LIN {X -29.370,Y -38.034,Z -132.609,A -90.000,B 90.000,C 0.000} C_DIS
LIN {X -29.590,Y -38.047,Z -132.219,A -90.000,B 90.000,C 0.000} C_DIS
LIN {X -30.207,Y -38.094,Z -131.099,A -90.000,B 90.000,C 0.000} C_DIS
LIN {X -30.398,Y -38.104,Z -130.742,A -90.000,B 90.000,C 0.000} C_DIS
LIN {X -30.507,Y -38.105,Z -130.533,A -90.000,B 90.000,C 0.000} C_DIS
LIN {X -31.312,Y -38.134,Z -128.926,A -90.000,B 90.000,C 0.000} C_DIS
LIN {X -31.541,Y -38.149,Z -128.454,A -90.000,B 90.000,C 0.000} C_DIS
LIN {X -31.849,Y -38.162,Z -127.810,A -90.000,B 90.000,C 0.000} C_DIS
LIN {X -31.967,Y -38.158,Z -127.548,A -90.000,B 90.000,C 0.000} C_DIS
LIN {X -32.731,Y -38.149,Z -125.792,A -90.000,B 90.000,C 0.000} C_DIS
LIN {X -32.828,Y -38.153,Z -125.553,A -90.000,B 90.000,C 0.000} C_DIS
LIN {X -32.982,Y -38.158,Z -125.157,A -90.000,B 90.000,C 0.000} C_DIS
LIN {X -33.082,Y -38.156,Z -124.892,A -90.000,B 90.000,C 0.000} C_DIS
LIN {X -33.162,Y -38.156,Z -124.675,A -90.000,B 90.000,C 0.000} C_DIS
LIN {X -33.245,Y -38.158,Z -124.435,A -90.000,B 90.000,C 0.000} C_DIS
LIN {X -33.570,Y -38.186,Z -123.415,A -90.000,B 90.000,C 0.000} C_DIS
LIN {X -33.902,Y -38.165,Z -122.569,A -90.000,B 90.000,C 0.000} C_DIS
LIN {X -33.950,Y -38.158,Z -122.440,A -90.000,B 90.000,C 0.000} C_DIS
LIN {X -34.013,Y -38.152,Z -122.276,A -90.000,B 90.000,C 0.000} C_DIS
LIN {X -34.135,Y -38.149,Z -121.934,A -90.000,B 90.000,C 0.000} C_DIS
LIN {X -34.194,Y -38.146,Z -121.753,A -90.000,B 90.000,C 0.000} C_DIS
LIN {X -34.258,Y -38.149,Z -121.536,A -90.000,B 90.000,C 0.000} C_DIS
LIN {X -34.518,Y -38.199,Z -120.499,A -90.000,B 90.000,C 0.000} C_DIS
LIN {X -34.562,Y -38.205,Z -120.316,A -90.000,B 90.000,C 0.000} C_DIS
LIN {X -34.581,Y -38.205,Z -120.229,A -90.000,B 90.000,C 0.000} C_DIS
LIN {X -34.750,Y -38.174,Z -119.659,A -90.000,B 90.000,C 0.000} C_DIS
LIN {X -34.930,Y -38.136,Z -119.039,A -90.000,B 90.000,C 0.000} C_DIS
LIN {X -34.971,Y -38.131,Z -118.875,A -90.000,B 90.000,C 0.000} C_DIS
LIN {X -34.998,Y -38.131,Z -118.751,A -90.000,B 90.000,C 0.000} C_DIS
LIN {X -35.069,Y -38.139,Z -118.462,A -90.000,B 90.000,C 0.000} C_DIS
LIN {X -35.272,Y -38.134,Z -117.766,A -90.000,B 90.000,C 0.000} C_DIS
LIN {X -35.322,Y -38.134,Z -117.585,A -90.000,B 90.000,C 0.000} C_DIS
LIN {X -35.400,Y -38.138,Z -117.219,A -90.000,B 90.000,C 0.000} C_DIS
LIN {X -35.446,Y -38.134,Z -116.963,A -90.000,B 90.000,C 0.000} C_DIS
LIN {X -35.540,Y -38.146,Z -116.520,A -90.000,B 90.000,C 0.000} C_DIS
LIN {X -35.611,Y -38.152,Z -116.171,A -90.000,B 90.000,C 0.000} C_DIS
LIN {X -35.725,Y -38.149,Z -115.614,A -90.000,B 90.000,C 0.000} C_DIS
LIN {X -35.750,Y -38.152,Z -115.472,A -90.000,B 90.000,C 0.000} C_DIS
LIN {X -35.834,Y -38.177,Z -114.889,A -90.000,B 90.000,C 0.000} C_DIS
LIN {X -35.887,Y -38.183,Z -114.459,A -90.000,B 90.000,C 0.000} C_DIS
LIN {X -36.126,Y -38.076,Z -112.938,A -90.000,B 90.000,C 0.000} C_DIS
LIN {X -36.182,Y -38.065,Z -112.617,A -90.000,B 90.000,C 0.000} C_DIS
LIN {X -36.199,Y -38.064,Z -112.499,A -90.000,B 90.000,C 0.000} C_DIS
LIN {X -36.214,Y -38.068,Z -112.354,A -90.000,B 90.000,C 0.000} C_DIS
LIN {X -36.251,Y -38.084,Z -111.934,A -90.000,B 90.000,C 0.000} C_DIS
LIN {X -36.282,Y -38.119,Z -111.373,A -90.000,B 90.000,C 0.000} C_DIS
LIN {X -36.295,Y -38.134,Z -111.034,A -90.000,B 90.000,C 0.000} C_DIS
LIN {X -36.296,Y -38.131,Z -110.722,A -90.000,B 90.000,C 0.000} C_DIS
LIN {X -36.288,Y -38.131,Z -110.115,A -90.000,B 90.000,C 0.000} C_DIS
LIN {X -36.294,Y -38.123,Z -109.819,A -90.000,B 90.000,C 0.000} C_DIS
LIN {X -36.294,Y -38.121,Z -109.575,A -90.000,B 90.000,C 0.000} C_DIS
LIN {X -36.288,Y -38.111,Z -109.292,A -90.000,B 90.000,C 0.000} C_DIS
LIN {X -36.281,Y -38.110,Z -109.154,A -90.000,B 90.000,C 0.000} C_DIS
LIN {X -36.263,Y -38.114,Z -108.902,A -90.000,B 90.000,C 0.000} C_DIS
LIN {X -36.234,Y -38.131,Z -108.455,A -90.000,B 90.000,C 0.000} C_DIS
LIN {X -36.217,Y -38.129,Z -108.275,A -90.000,B 90.000,C 0.000} C_DIS
LIN {X -36.200,Y -38.123,Z -108.047,A -90.000,B 90.000,C 0.000} C_DIS
LIN {X -36.088,Y -38.061,Z -106.817,A -90.000,B 90.000,C 0.000} C_DIS
LIN {X -36.081,Y -38.058,Z -106.727,A -90.000,B 90.000,C 0.000} C_DIS
LIN {X -36.038,Y -38.050,Z -106.281,A -90.000,B 90.000,C 0.000} C_DIS
LIN {X -36.018,Y -38.051,Z -106.126,A -90.000,B 90.000,C 0.000} C_DIS
LIN {X -35.925,Y -38.071,Z -105.532,A -90.000,B 90.000,C 0.000} C_DIS
LIN {X -35.871,Y -38.073,Z -105.235,A -90.000,B 90.000,C 0.000} C_DIS
LIN {X -35.704,Y -38.058,Z -104.390,A -90.000,B 90.000,C 0.000} C_DIS
LIN {X -35.642,Y -38.057,Z -104.114,A -90.000,B 90.000,C 0.000} C_DIS
LIN {X -35.588,Y -38.052,Z -103.880,A -90.000,B 90.000,C 0.000} C_DIS
LIN {X -35.548,Y -38.048,Z -103.705,A -90.000,B 90.000,C 0.000} C_DIS
LIN {X -35.328,Y -38.051,Z -102.848,A -90.000,B 90.000,C 0.000} C_DIS
LIN {X -35.183,Y -38.044,Z -102.313,A -90.000,B 90.000,C 0.000} C_DIS
LIN {X -34.966,Y -38.023,Z -101.474,A -90.000,B 90.000,C 0.000} C_DIS
LIN {X -34.772,Y -38.008,Z -100.758,A -90.000,B 90.000,C 0.000} C_DIS
LIN {X -34.674,Y -37.996,Z -100.376,A -90.000,B 90.000,C 0.000} C_DIS
LIN {X -34.582,Y -37.990,Z -100.004,A -90.000,B 90.000,C 0.000} C_DIS
LIN {X -34.433,Y -37.969,Z -99.437,A -90.000,B 90.000,C 0.000} C_DIS
LIN {X -34.339,Y -37.964,Z -99.109,A -90.000,B 90.000,C 0.000} C_DIS
LIN {X -34.237,Y -37.962,Z -98.761,A -90.000,B 90.000,C 0.000} C_DIS
LIN {X -34.128,Y -37.965,Z -98.376,A -90.000,B 90.000,C 0.000} C_DIS
LIN {X -33.923,Y -37.959,Z -97.689,A -90.000,B 90.000,C 0.000} C_DIS
LIN {X -33.862,Y -37.961,Z -97.470,A -90.000,B 90.000,C 0.000} C_DIS
LIN {X -33.743,Y -37.968,Z -97.056,A -90.000,B 90.000,C 0.000} C_DIS
LIN {X -33.704,Y -37.968,Z -96.908,A -90.000,B 90.000,C 0.000} C_DIS
LIN {X -33.649,Y -37.972,Z -96.719,A -90.000,B 90.000,C 0.000} C_DIS
LIN {X -33.580,Y -37.978,Z -96.489,A -90.000,B 90.000,C 0.000} C_DIS
LIN {X -33.507,Y -37.990,Z -96.233,A -90.000,B 90.000,C 0.000} C_DIS
LIN {X -33.465,Y -37.995,Z -96.088,A -90.000,B 90.000,C 0.000} C_DIS
LIN {X -33.404,Y -37.996,Z -95.875,A -90.000,B 90.000,C 0.000} C_DIS
LIN {X -33.339,Y -38.056,Z -95.468,A -90.000,B 90.000,C 0.000} C_DIS
LIN {X -33.319,Y -38.083,Z -95.323,A -90.000,B 90.000,C 0.000} C_DIS
LIN {X -33.245,Y -38.178,Z -94.834,A -90.000,B 90.000,C 0.000} C_DIS
LIN {X -33.197,Y -38.234,Z -94.546,A -90.000,B 90.000,C 0.000} C_DIS
LIN {X -33.125,Y -38.309,Z -94.171,A -90.000,B 90.000,C 0.000} C_DIS
LIN {X -33.034,Y -38.389,Z -93.783,A -90.000,B 90.000,C 0.000} C_DIS
LIN {X -32.956,Y -38.440,Z -93.489,A -90.000,B 90.000,C 0.000} C_DIS
LIN {X -32.805,Y -38.538,Z -92.936,A -90.000,B 90.000,C 0.000} C_DIS
LIN {X -32.662,Y -38.640,Z -92.322,A -90.000,B 90.000,C 0.000} C_DIS
LIN {X -32.562,Y -38.708,Z -91.928,A -90.000,B 90.000,C 0.000} C_DIS
LIN {X -32.532,Y -38.727,Z -91.826,A -90.000,B 90.000,C 0.000} C_DIS
LIN {X -32.500,Y -38.746,Z -91.724,A -90.000,B 90.000,C 0.000} C_DIS
LIN {X -32.485,Y -38.753,Z -91.679,A -90.000,B 90.000,C 0.000} C_DIS
LIN {X -32.402,Y -38.790,Z -91.376,A -90.000,B 90.000,C 0.000} C_DIS
LIN {X -32.313,Y -38.822,Z -91.059,A -90.000,B 90.000,C 0.000} C_DIS
LIN {X -32.092,Y -38.896,Z -90.344,A -90.000,B 90.000,C 0.000} C_DIS
LIN {X -32.085,Y -38.899,Z -90.305,A -90.000,B 90.000,C 0.000} C_DIS
LIN {X -32.084,Y -38.900,Z -90.286,A -90.000,B 90.000,C 0.000} C_DIS
LIN {X -32.064,Y -38.920,Z -89.990,A -90.000,B 90.000,C 0.000} C_DIS
LIN {X -32.032,Y -38.938,Z -89.747,A -90.000,B 90.000,C 0.000} C_DIS
LIN {X -31.910,Y -38.991,Z -89.128,A -90.000,B 90.000,C 0.000} C_DIS
LIN {X -31.879,Y -38.997,Z -88.974,A -90.000,B 90.000,C 0.000} C_DIS
LIN {X -31.743,Y -39.003,Z -88.329,A -90.000,B 90.000,C 0.000} C_DIS
LIN {X -31.565,Y -39.013,Z -87.526,A -90.000,B 90.000,C 0.000} C_DIS
LIN {X -31.524,Y -39.015,Z -87.334,A -90.000,B 90.000,C 0.000} C_DIS
LIN {X -31.485,Y -39.018,Z -87.166,A -90.000,B 90.000,C 0.000} C_DIS
LIN {X -31.438,Y -39.022,Z -87.019,A -90.000,B 90.000,C 0.000} C_DIS
LIN {X -31.378,Y -39.028,Z -86.868,A -90.000,B 90.000,C 0.000} C_DIS
LIN {X -31.347,Y -39.030,Z -86.804,A -90.000,B 90.000,C 0.000} C_DIS
LIN {X -31.307,Y -39.033,Z -86.726,A -90.000,B 90.000,C 0.000} C_DIS
LIN {X -31.215,Y -39.034,Z -86.557,A -90.000,B 90.000,C 0.000} C_DIS
LIN {X -30.944,Y -39.030,Z -86.124,A -90.000,B 90.000,C 0.000} C_DIS
LIN {X -30.545,Y -39.018,Z -85.401,A -90.000,B 90.000,C 0.000} C_DIS
LIN {X -30.121,Y -39.010,Z -84.656,A -90.000,B 90.000,C 0.000} C_DIS
LIN {X -30.034,Y -39.004,Z -84.508,A -90.000,B 90.000,C 0.000} C_DIS
LIN {X -29.948,Y -38.997,Z -84.382,A -90.000,B 90.000,C 0.000} C_DIS
LIN {X -29.903,Y -38.995,Z -84.323,A -90.000,B 90.000,C 0.000} C_DIS
LIN {X -29.678,Y -38.984,Z -84.066,A -90.000,B 90.000,C 0.000} C_DIS
LIN {X -29.090,Y -38.961,Z -83.456,A -90.000,B 90.000,C 0.000} C_DIS
LIN {X -28.750,Y -38.953,Z -83.123,A -90.000,B 90.000,C 0.000} C_DIS
LIN {X -28.382,Y -38.933,Z -82.672,A -90.000,B 90.000,C 0.000} C_DIS
LIN {X -28.290,Y -38.925,Z -82.561,A -90.000,B 90.000,C 0.000} C_DIS
LIN {X -28.086,Y -38.900,Z -82.315,A -90.000,B 90.000,C 0.000} C_DIS
LIN {X -28.031,Y -38.894,Z -82.252,A -90.000,B 90.000,C 0.000} C_DIS
LIN {X -27.808,Y -38.873,Z -82.017,A -90.000,B 90.000,C 0.000} C_DIS
LIN {X -27.730,Y -38.867,Z -81.941,A -90.000,B 90.000,C 0.000} C_DIS
LIN {X -27.302,Y -38.834,Z -81.540,A -90.000,B 90.000,C 0.000} C_DIS
LIN {X -26.767,Y -38.778,Z -80.939,A -90.000,B 90.000,C 0.000} C_DIS
LIN {X -26.416,Y -38.748,Z -80.544,A -90.000,B 90.000,C 0.000} C_DIS
LIN {X -26.257,Y -38.732,Z -80.352,A -90.000,B 90.000,C 0.000} C_DIS
LIN {X -26.136,Y -38.713,Z -80.210,A -90.000,B 90.000,C 0.000} C_DIS
LIN {X -26.030,Y -38.696,Z -80.088,A -90.000,B 90.000,C 0.000} C_DIS
LIN {X -25.812,Y -38.663,Z -79.854,A -90.000,B 90.000,C 0.000} C_DIS
LIN {X -24.861,Y -38.532,Z -78.886,A -90.000,B 90.000,C 0.000} C_DIS
LIN {X -24.274,Y -38.484,Z -78.275,A -90.000,B 90.000,C 0.000} C_DIS
LIN {X -24.019,Y -38.464,Z -78.012,A -90.000,B 90.000,C 0.000} C_DIS
LIN {X -23.833,Y -38.441,Z -77.829,A -90.000,B 90.000,C 0.000} C_DIS
LIN {X -23.570,Y -38.424,Z -77.561,A -90.000,B 90.000,C 0.000} C_DIS
LIN {X -23.506,Y -38.422,Z -77.502,A -90.000,B 90.000,C 0.000} C_DIS
LIN {X -22.883,Y -38.410,Z -76.951,A -90.000,B 90.000,C 0.000} C_DIS
LIN {X -21.992,Y -38.423,Z -76.142,A -90.000,B 90.000,C 0.000} C_DIS
LIN {X -21.889,Y -38.426,Z -76.053,A -90.000,B 90.000,C 0.000} C_DIS
LIN {X -21.703,Y -38.428,Z -75.895,A -90.000,B 90.000,C 0.000} C_DIS
LIN {X -21.556,Y -38.430,Z -75.777,A -90.000,B 90.000,C 0.000} C_DIS
LIN {X -21.246,Y -38.428,Z -75.536,A -90.000,B 90.000,C 0.000} C_DIS
LIN {X -21.142,Y -38.429,Z -75.460,A -90.000,B 90.000,C 0.000} C_DIS
LIN {X -20.706,Y -38.427,Z -75.155,A -90.000,B 90.000,C 0.000} C_DIS
LIN {X -20.564,Y -38.428,Z -75.061,A -90.000,B 90.000,C 0.000} C_DIS
LIN {X -20.428,Y -38.432,Z -74.977,A -90.000,B 90.000,C 0.000} C_DIS
LIN {X -20.223,Y -38.438,Z -74.852,A -90.000,B 90.000,C 0.000} C_DIS
LIN {X -19.490,Y -38.474,Z -74.435,A -90.000,B 90.000,C 0.000} C_DIS
LIN {X -19.405,Y -38.480,Z -74.389,A -90.000,B 90.000,C 0.000} C_DIS
LIN {X -19.147,Y -38.492,Z -74.264,A -90.000,B 90.000,C 0.000} C_DIS
LIN {X -18.935,Y -38.498,Z -74.165,A -90.000,B 90.000,C 0.000} C_DIS
LIN {X -18.780,Y -38.498,Z -74.093,A -90.000,B 90.000,C 0.000} C_DIS
LIN {X -18.579,Y -38.501,Z -74.009,A -90.000,B 90.000,C 0.000} C_DIS
LIN {X -18.282,Y -38.502,Z -73.889,A -90.000,B 90.000,C 0.000} C_DIS
LIN {X -18.130,Y -38.494,Z -73.832,A -90.000,B 90.000,C 0.000} C_DIS
LIN {X -17.614,Y -38.473,Z -73.648,A -90.000,B 90.000,C 0.000} C_DIS
LIN {X -17.496,Y -38.470,Z -73.609,A -90.000,B 90.000,C 0.000} C_DIS
LIN {X -17.399,Y -38.469,Z -73.581,A -90.000,B 90.000,C 0.000} C_DIS
LIN {X -17.194,Y -38.464,Z -73.523,A -90.000,B 90.000,C 0.000} C_DIS
LIN {X -16.402,Y -38.442,Z -73.304,A -90.000,B 90.000,C 0.000} C_DIS
LIN {X -16.126,Y -38.426,Z -73.234,A -90.000,B 90.000,C 0.000} C_DIS
LIN {X -15.986,Y -38.419,Z -73.201,A -90.000,B 90.000,C 0.000} C_DIS
LIN {X -15.624,Y -38.406,Z -73.125,A -90.000,B 90.000,C 0.000} C_DIS
LIN {X -15.502,Y -38.403,Z -73.107,A -90.000,B 90.000,C 0.000} C_DIS
LIN {X -15.182,Y -38.397,Z -73.066,A -90.000,B 90.000,C 0.000} C_DIS
LIN {X -14.881,Y -38.397,Z -73.037,A -90.000,B 90.000,C 0.000} C_DIS
LIN {X -14.525,Y -38.400,Z -73.009,A -90.000,B 90.000,C 0.000} C_DIS
LIN {X -14.442,Y -38.401,Z -73.004,A -90.000,B 90.000,C 0.000} C_DIS
LIN {X -13.919,Y -38.416,Z -72.983,A -90.000,B 90.000,C 0.000} C_DIS
LIN {X -13.429,Y -38.425,Z -72.965,A -90.000,B 90.000,C 0.000} C_DIS
LIN {X -12.736,Y -38.408,Z -72.956,A -90.000,B 90.000,C 0.000} C_DIS
LIN {X -12.449,Y -38.404,Z -72.957,A -90.000,B 90.000,C 0.000} C_DIS
LIN {X -11.202,Y -38.373,Z -72.976,A -90.000,B 90.000,C 0.000} C_DIS
LIN {X -10.399,Y -38.374,Z -73.025,A -90.000,B 90.000,C 0.000} C_DIS
LIN {X -10.048,Y -38.373,Z -73.051,A -90.000,B 90.000,C 0.000} C_DIS
LIN {X -9.056,Y -38.353,Z -73.141,A -90.000,B 90.000,C 0.000} C_DIS
LIN {X -8.105,Y -38.335,Z -73.228,A -90.000,B 90.000,C 0.000} C_DIS
LIN {X -7.181,Y -38.331,Z -73.334,A -90.000,B 90.000,C 0.000} C_DIS
LIN {X -7.058,Y -38.333,Z -73.351,A -90.000,B 90.000,C 0.000} C_DIS
LIN {X -6.263,Y -38.354,Z -73.487,A -90.000,B 90.000,C 0.000} C_DIS
LIN {X -5.825,Y -38.354,Z -73.568,A -90.000,B 90.000,C 0.000} C_DIS
LIN {X -4.312,Y -38.360,Z -73.847,A -90.000,B 90.000,C 0.000} C_DIS
LIN {X -2.722,Y -38.350,Z -74.131,A -90.000,B 90.000,C 0.000} C_DIS
LIN {X -2.009,Y -38.363,Z -74.278,A -90.000,B 90.000,C 0.000} C_DIS
LIN {X -1.453,Y -38.363,Z -74.401,A -90.000,B 90.000,C 0.000} C_DIS
LIN {X -0.231,Y -38.356,Z -74.660,A -90.000,B 90.000,C 0.000} C_DIS
LIN {X 0.946,Y -38.361,Z -74.904,A -90.000,B 90.000,C 0.000} C_DIS
LIN {X 1.526,Y -38.366,Z -75.029,A -90.000,B 90.000,C 0.000} C_DIS
LIN {X 1.757,Y -38.366,Z -75.075,A -90.000,B 90.000,C 0.000} C_DIS
LIN {X 2.460,Y -38.379,Z -75.235,A -90.000,B 90.000,C 0.000} C_DIS
LIN {X 2.784,Y -38.390,Z -75.306,A -90.000,B 90.000,C 0.000} C_DIS
LIN {X 4.308,Y -38.416,Z -75.659,A -90.000,B 90.000,C 0.000} C_DIS
LIN {X 5.039,Y -38.423,Z -75.816,A -90.000,B 90.000,C 0.000} C_DIS
LIN {X 6.224,Y -38.451,Z -76.062,A -90.000,B 90.000,C 0.000} C_DIS
LIN {X 6.707,Y -38.468,Z -76.174,A -90.000,B 90.000,C 0.000} C_DIS
LIN {X 7.203,Y -38.510,Z -76.278,A -90.000,B 90.000,C 0.000} C_DIS
LIN {X 8.101,Y -38.570,Z -76.471,A -90.000,B 90.000,C 0.000} C_DIS
LIN {X 8.376,Y -38.586,Z -76.521,A -90.000,B 90.000,C 0.000} C_DIS
LIN {X 8.626,Y -38.603,Z -76.565,A -90.000,B 90.000,C 0.000} C_DIS
LIN {X 9.269,Y -38.677,Z -76.669,A -90.000,B 90.000,C 0.000} C_DIS
LIN {X 9.419,Y -38.693,Z -76.690,A -90.000,B 90.000,C 0.000} C_DIS
LIN {X 10.343,Y -38.809,Z -76.812,A -90.000,B 90.000,C 0.000} C_DIS
LIN {X 10.515,Y -38.831,Z -76.841,A -90.000,B 90.000,C 0.000} C_DIS
LIN {X 10.822,Y -38.880,Z -76.898,A -90.000,B 90.000,C 0.000} C_DIS
LIN {X 11.012,Y -38.911,Z -76.933,A -90.000,B 90.000,C 0.000} C_DIS
LIN {X 11.634,Y -38.999,Z -76.917,A -90.000,B 90.000,C 0.000} C_DIS
LIN {X 11.711,Y -39.009,Z -76.910,A -90.000,B 90.000,C 0.000} C_DIS
LIN {X 11.718,Y -39.009,Z -76.906,A -90.000,B 90.000,C 0.000} C_DIS
LIN {X 11.753,Y -39.010,Z -76.863,A -90.000,B 90.000,C 0.000} C_DIS
LIN {X 12.009,Y -39.013,Z -76.565,A -90.000,B 90.000,C 0.000} C_DIS
LIN {X 12.309,Y -39.010,Z -76.219,A -90.000,B 90.000,C 0.000} C_DIS
LIN {X 12.640,Y -39.010,Z -75.869,A -90.000,B 90.000,C 0.000} C_DIS
LIN {X 12.774,Y -39.011,Z -75.732,A -90.000,B 90.000,C 0.000} C_DIS
LIN {X 12.860,Y -39.012,Z -75.647,A -90.000,B 90.000,C 0.000} C_DIS
LIN {X 12.948,Y -39.013,Z -75.571,A -90.000,B 90.000,C 0.000} C_DIS
LIN {X 12.996,Y -39.014,Z -75.532,A -90.000,B 90.000,C 0.000} C_DIS
LIN {X 13.082,Y -39.013,Z -75.470,A -90.000,B 90.000,C 0.000} C_DIS
LIN {X 13.290,Y -39.012,Z -75.335,A -90.000,B 90.000,C 0.000} C_DIS
LIN {X 13.745,Y -38.978,Z -75.050,A -90.000,B 90.000,C 0.000} C_DIS
LIN {X 13.871,Y -38.960,Z -74.973,A -90.000,B 90.000,C 0.000} C_DIS
LIN {X 13.974,Y -38.941,Z -74.915,A -90.000,B 90.000,C 0.000} C_DIS
LIN {X 14.122,Y -38.917,Z -74.836,A -90.000,B 90.000,C 0.000} C_DIS
LIN {X 14.247,Y -38.899,Z -74.775,A -90.000,B 90.000,C 0.000} C_DIS
LIN {X 14.306,Y -38.891,Z -74.750,A -90.000,B 90.000,C 0.000} C_DIS
LIN {X 14.416,Y -38.879,Z -74.709,A -90.000,B 90.000,C 0.000} C_DIS
LIN {X 14.656,Y -38.858,Z -74.642,A -90.000,B 90.000,C 0.000} C_DIS
LIN {X 14.591,Y -38.801,Z -74.423,A -90.000,B 90.000,C 0.000} C_DIS
LIN {X 14.553,Y -38.752,Z -74.238,A -90.000,B 90.000,C 0.000} C_DIS
LIN {X 14.501,Y -38.653,Z -73.861,A -90.000,B 90.000,C 0.000} C_DIS
LIN {X 14.469,Y -38.576,Z -73.577,A -90.000,B 90.000,C 0.000} C_DIS
LIN {X 14.439,Y -38.482,Z -73.252,A -90.000,B 90.000,C 0.000} C_DIS
LIN {X 14.415,Y -38.384,Z -72.916,A -90.000,B 90.000,C 0.000} C_DIS
LIN {X 14.414,Y -38.346,Z -72.793,A -90.000,B 90.000,C 0.000} C_DIS
LIN {X 14.429,Y -38.244,Z -72.478,A -90.000,B 90.000,C 0.000} C_DIS
LIN {X 14.462,Y -38.115,Z -72.092,A -90.000,B 90.000,C 0.000} C_DIS
LIN {X 14.448,Y -38.119,Z -71.998,A -90.000,B 90.000,C 0.000} C_DIS
LIN {X 14.413,Y -38.137,Z -71.633,A -90.000,B 90.000,C 0.000} C_DIS
LIN {X 14.405,Y -38.141,Z -71.490,A -90.000,B 90.000,C 0.000} C_DIS
LIN {X 14.402,Y -38.158,Z -71.246,A -90.000,B 90.000,C 0.000} C_DIS
LIN {X 14.409,Y -38.187,Z -70.924,A -90.000,B 90.000,C 0.000} C_DIS
LIN {X 14.419,Y -38.191,Z -70.789,A -90.000,B 90.000,C 0.000} C_DIS
LIN {X 14.441,Y -38.202,Z -70.628,A -90.000,B 90.000,C 0.000} C_DIS
LIN {X 14.478,Y -38.223,Z -70.407,A -90.000,B 90.000,C 0.000} C_DIS
LIN {X 14.518,Y -38.239,Z -70.206,A -90.000,B 90.000,C 0.000} C_DIS
LIN {X 14.550,Y -38.253,Z -70.080,A -90.000,B 90.000,C 0.000} C_DIS
LIN {X 14.630,Y -38.269,Z -69.844,A -90.000,B 90.000,C 0.000} C_DIS
LIN {X 14.707,Y -38.287,Z -69.638,A -90.000,B 90.000,C 0.000} C_DIS
LIN {X 14.823,Y -38.307,Z -69.382,A -90.000,B 90.000,C 0.000} C_DIS
LIN {X 14.897,Y -38.323,Z -69.232,A -90.000,B 90.000,C 0.000} C_DIS
LIN {X 15.007,Y -38.345,Z -69.033,A -90.000,B 90.000,C 0.000} C_DIS
LIN {X 15.096,Y -38.357,Z -68.883,A -90.000,B 90.000,C 0.000} C_DIS
LIN {X 15.180,Y -38.368,Z -68.765,A -90.000,B 90.000,C 0.000} C_DIS
LIN {X 15.317,Y -38.389,Z -68.590,A -90.000,B 90.000,C 0.000} C_DIS
LIN {X 15.404,Y -38.393,Z -68.487,A -90.000,B 90.000,C 0.000} C_DIS
LIN {X 15.523,Y -38.402,Z -68.356,A -90.000,B 90.000,C 0.000} C_DIS
LIN {X 15.544,Y -38.405,Z -68.335,A -90.000,B 90.000,C 0.000} C_DIS
LIN {X 15.786,Y -38.416,Z -68.123,A -90.000,B 90.000,C 0.000} C_DIS
LIN {X 15.840,Y -38.415,Z -68.078,A -90.000,B 90.000,C 0.000} C_DIS
LIN {X 16.042,Y -38.416,Z -67.931,A -90.000,B 90.000,C 0.000} C_DIS
LIN {X 16.089,Y -38.418,Z -67.901,A -90.000,B 90.000,C 0.000} C_DIS
LIN {X 16.393,Y -38.411,Z -67.724,A -90.000,B 90.000,C 0.000} C_DIS
LIN {X 16.477,Y -38.405,Z -67.683,A -90.000,B 90.000,C 0.000} C_DIS
LIN {X 16.551,Y -38.402,Z -67.651,A -90.000,B 90.000,C 0.000} C_DIS
LIN {X 16.713,Y -38.399,Z -67.586,A -90.000,B 90.000,C 0.000} C_DIS
LIN {X 16.785,Y -38.393,Z -67.560,A -90.000,B 90.000,C 0.000} C_DIS
LIN {X 16.894,Y -38.387,Z -67.520,A -90.000,B 90.000,C 0.000} C_DIS
LIN {X 17.067,Y -38.382,Z -67.462,A -90.000,B 90.000,C 0.000} C_DIS
LIN {X 17.162,Y -38.384,Z -67.437,A -90.000,B 90.000,C 0.000} C_DIS
LIN {X 17.282,Y -38.380,Z -67.396,A -90.000,B 90.000,C 0.000} C_DIS
LIN {X 17.611,Y -38.359,Z -67.292,A -90.000,B 90.000,C 0.000} C_DIS
LIN {X 17.753,Y -38.346,Z -67.262,A -90.000,B 90.000,C 0.000} C_DIS
LIN {X 17.995,Y -38.326,Z -67.217,A -90.000,B 90.000,C 0.000} C_DIS
LIN {X 18.152,Y -38.305,Z -67.196,A -90.000,B 90.000,C 0.000} C_DIS
LIN {X 18.326,Y -38.285,Z -67.180,A -90.000,B 90.000,C 0.000} C_DIS
LIN {X 18.412,Y -38.276,Z -67.179,A -90.000,B 90.000,C 0.000} C_DIS
LIN {X 18.685,Y -38.244,Z -67.180,A -90.000,B 90.000,C 0.000} C_DIS
LIN {X 18.825,Y -38.228,Z -67.184,A -90.000,B 90.000,C 0.000} C_DIS
LIN {X 18.991,Y -38.210,Z -67.202,A -90.000,B 90.000,C 0.000} C_DIS
LIN {X 19.348,Y -38.178,Z -67.249,A -90.000,B 90.000,C 0.000} C_DIS
LIN {X 19.590,Y -38.153,Z -67.286,A -90.000,B 90.000,C 0.000} C_DIS
LIN {X 19.716,Y -38.140,Z -67.310,A -90.000,B 90.000,C 0.000} C_DIS
LIN {X 19.876,Y -38.130,Z -67.349,A -90.000,B 90.000,C 0.000} C_DIS
LIN {X 20.044,Y -38.222,Z -67.322,A -90.000,B 90.000,C 0.000} C_DIS
LIN {X 20.235,Y -38.315,Z -67.308,A -90.000,B 90.000,C 0.000} C_DIS
LIN {X 20.417,Y -38.406,Z -67.305,A -90.000,B 90.000,C 0.000} C_DIS
LIN {X 20.542,Y -38.468,Z -67.308,A -90.000,B 90.000,C 0.000} C_DIS
LIN {X 20.589,Y -38.470,Z -67.241,A -90.000,B 90.000,C 0.000} C_DIS
LIN {X 20.671,Y -38.472,Z -67.138,A -90.000,B 90.000,C 0.000} C_DIS
LIN {X 20.816,Y -38.479,Z -66.970,A -90.000,B 90.000,C 0.000} C_DIS
LIN {X 20.967,Y -38.480,Z -66.810,A -90.000,B 90.000,C 0.000} C_DIS
LIN {X 21.072,Y -38.478,Z -66.717,A -90.000,B 90.000,C 0.000} C_DIS
LIN {X 21.210,Y -38.478,Z -66.601,A -90.000,B 90.000,C 0.000} C_DIS
LIN {X 21.315,Y -38.473,Z -66.524,A -90.000,B 90.000,C 0.000} C_DIS
LIN {X 21.468,Y -38.465,Z -66.418,A -90.000,B 90.000,C 0.000} C_DIS
LIN {X 21.639,Y -38.458,Z -66.317,A -90.000,B 90.000,C 0.000} C_DIS
LIN {X 21.765,Y -38.448,Z -66.251,A -90.000,B 90.000,C 0.000} C_DIS
LIN {X 21.945,Y -38.438,Z -66.167,A -90.000,B 90.000,C 0.000} C_DIS
LIN {X 22.061,Y -38.426,Z -66.121,A -90.000,B 90.000,C 0.000} C_DIS
LIN {X 22.255,Y -38.410,Z -66.053,A -90.000,B 90.000,C 0.000} C_DIS
LIN {X 22.359,Y -38.397,Z -66.026,A -90.000,B 90.000,C 0.000} C_DIS
LIN {X 22.564,Y -38.374,Z -65.979,A -90.000,B 90.000,C 0.000} C_DIS
LIN {X 22.680,Y -38.360,Z -65.956,A -90.000,B 90.000,C 0.000} C_DIS
LIN {X 22.823,Y -38.342,Z -65.932,A -90.000,B 90.000,C 0.000} C_DIS
LIN {X 23.032,Y -38.313,Z -65.901,A -90.000,B 90.000,C 0.000} C_DIS
LIN {X 23.183,Y -38.295,Z -65.886,A -90.000,B 90.000,C 0.000} C_DIS
LIN {X 23.320,Y -38.281,Z -65.882,A -90.000,B 90.000,C 0.000} C_DIS
LIN {X 23.627,Y -38.241,Z -65.885,A -90.000,B 90.000,C 0.000} C_DIS
LIN {X 23.755,Y -38.221,Z -65.897,A -90.000,B 90.000,C 0.000} C_DIS
LIN {X 24.325,Y -38.145,Z -65.966,A -90.000,B 90.000,C 0.000} C_DIS
LIN {X 24.623,Y -38.093,Z -66.027,A -90.000,B 90.000,C 0.000} C_DIS
LIN {X 24.797,Y -38.065,Z -66.066,A -90.000,B 90.000,C 0.000} C_DIS
LIN {X 24.822,Y -38.073,Z -66.064,A -90.000,B 90.000,C 0.000} C_DIS
LIN {X 24.943,Y -38.111,Z -66.055,A -90.000,B 90.000,C 0.000} C_DIS
LIN {X 25.149,Y -38.178,Z -66.048,A -90.000,B 90.000,C 0.000} C_DIS
LIN {X 25.259,Y -38.213,Z -66.047,A -90.000,B 90.000,C 0.000} C_DIS
LIN {X 25.458,Y -38.275,Z -66.052,A -90.000,B 90.000,C 0.000} C_DIS
LIN {X 25.679,Y -38.344,Z -66.069,A -90.000,B 90.000,C 0.000} C_DIS
LIN {X 25.999,Y -38.442,Z -66.103,A -90.000,B 90.000,C 0.000} C_DIS
LIN {X 26.250,Y -38.520,Z -66.135,A -90.000,B 90.000,C 0.000} C_DIS
LIN {X 26.416,Y -38.572,Z -66.164,A -90.000,B 90.000,C 0.000} C_DIS
LIN {X 26.636,Y -38.571,Z -66.001,A -90.000,B 90.000,C 0.000} C_DIS
LIN {X 26.646,Y -38.536,Z -65.890,A -90.000,B 90.000,C 0.000} C_DIS
LIN {X 26.681,Y -38.421,Z -65.538,A -90.000,B 90.000,C 0.000} C_DIS
LIN {X 26.731,Y -38.310,Z -65.199,A -90.000,B 90.000,C 0.000} C_DIS
LIN {X 26.742,Y -38.289,Z -65.141,A -90.000,B 90.000,C 0.000} C_DIS
LIN {X 26.782,Y -38.218,Z -64.959,A -90.000,B 90.000,C 0.000} C_DIS
LIN {X 26.846,Y -38.116,Z -64.694,A -90.000,B 90.000,C 0.000} C_DIS
LIN {X 26.910,Y -38.028,Z -64.462,A -90.000,B 90.000,C 0.000} C_DIS
LIN {X 26.943,Y -37.988,Z -64.355,A -90.000,B 90.000,C 0.000} C_DIS
LIN {X 27.012,Y -37.910,Z -64.145,A -90.000,B 90.000,C 0.000} C_DIS
LIN {X 27.069,Y -37.852,Z -63.991,A -90.000,B 90.000,C 0.000} C_DIS
LIN {X 27.125,Y -37.800,Z -63.852,A -90.000,B 90.000,C 0.000} C_DIS
LIN {X 27.191,Y -37.743,Z -63.699,A -90.000,B 90.000,C 0.000} C_DIS
LIN {X 27.226,Y -37.717,Z -63.627,A -90.000,B 90.000,C 0.000} C_DIS
LIN {X 27.297,Y -37.668,Z -63.488,A -90.000,B 90.000,C 0.000} C_DIS
LIN {X 27.379,Y -37.616,Z -63.338,A -90.000,B 90.000,C 0.000} C_DIS
LIN {X 27.457,Y -37.571,Z -63.221,A -90.000,B 90.000,C 0.000} C_DIS
LIN {X 27.548,Y -37.524,Z -63.096,A -90.000,B 90.000,C 0.000} C_DIS
LIN {X 27.521,Y -37.544,Z -62.796,A -90.000,B 90.000,C 0.000} C_DIS
LIN {X 27.499,Y -37.561,Z -62.517,A -90.000,B 90.000,C 0.000} C_DIS
LIN {X 27.472,Y -37.593,Z -62.124,A -90.000,B 90.000,C 0.000} C_DIS
LIN {X 27.452,Y -37.634,Z -61.769,A -90.000,B 90.000,C 0.000} C_DIS
LIN {X 27.453,Y -37.657,Z -61.507,A -90.000,B 90.000,C 0.000} C_DIS
LIN {X 27.461,Y -37.709,Z -60.992,A -90.000,B 90.000,C 0.000} C_DIS
LIN {X 27.485,Y -37.742,Z -60.595,A -90.000,B 90.000,C 0.000} C_DIS
LIN {X 27.536,Y -37.788,Z -60.131,A -90.000,B 90.000,C 0.000} C_DIS
LIN {X 27.558,Y -37.809,Z -59.964,A -90.000,B 90.000,C 0.000} C_DIS
LIN {X 27.662,Y -37.862,Z -59.513,A -90.000,B 90.000,C 0.000} C_DIS
LIN {X 27.765,Y -37.893,Z -59.193,A -90.000,B 90.000,C 0.000} C_DIS
LIN {X 27.889,Y -37.933,Z -58.835,A -90.000,B 90.000,C 0.000} C_DIS
LIN {X 27.944,Y -37.944,Z -58.698,A -90.000,B 90.000,C 0.000} C_DIS
LIN {X 27.977,Y -37.952,Z -58.624,A -90.000,B 90.000,C 0.000} C_DIS
LIN {X 28.149,Y -37.995,Z -58.285,A -90.000,B 90.000,C 0.000} C_DIS
LIN {X 28.213,Y -38.008,Z -58.169,A -90.000,B 90.000,C 0.000} C_DIS
LIN {X 28.286,Y -38.027,Z -58.047,A -90.000,B 90.000,C 0.000} C_DIS
LIN {X 28.487,Y -38.063,Z -57.737,A -90.000,B 90.000,C 0.000} C_DIS
LIN {X 28.564,Y -38.068,Z -57.634,A -90.000,B 90.000,C 0.000} C_DIS
LIN {X 28.640,Y -38.078,Z -57.542,A -90.000,B 90.000,C 0.000} C_DIS
LIN {X 28.728,Y -38.091,Z -57.441,A -90.000,B 90.000,C 0.000} C_DIS
LIN {X 28.832,Y -38.102,Z -57.328,A -90.000,B 90.000,C 0.000} C_DIS
LIN {X 28.926,Y -38.109,Z -57.230,A -90.000,B 90.000,C 0.000} C_DIS
LIN {X 29.033,Y -38.122,Z -57.128,A -90.000,B 90.000,C 0.000} C_DIS
LIN {X 29.093,Y -38.131,Z -57.075,A -90.000,B 90.000,C 0.000} C_DIS
LIN {X 29.383,Y -38.151,Z -56.846,A -90.000,B 90.000,C 0.000} C_DIS
LIN {X 29.574,Y -38.152,Z -56.716,A -90.000,B 90.000,C 0.000} C_DIS
LIN {X 29.697,Y -38.156,Z -56.637,A -90.000,B 90.000,C 0.000} C_DIS
LIN {X 29.908,Y -38.159,Z -56.523,A -90.000,B 90.000,C 0.000} C_DIS
LIN {X 30.022,Y -38.158,Z -56.462,A -90.000,B 90.000,C 0.000} C_DIS
LIN {X 30.128,Y -38.159,Z -56.410,A -90.000,B 90.000,C 0.000} C_DIS
LIN {X 30.241,Y -38.164,Z -56.360,A -90.000,B 90.000,C 0.000} C_DIS
LIN {X 30.564,Y -38.163,Z -56.243,A -90.000,B 90.000,C 0.000} C_DIS
LIN {X 30.605,Y -38.164,Z -56.229,A -90.000,B 90.000,C 0.000} C_DIS
LIN {X 30.661,Y -38.161,Z -56.213,A -90.000,B 90.000,C 0.000} C_DIS
LIN {X 30.711,Y -38.121,Z -56.147,A -90.000,B 90.000,C 0.000} C_DIS
LIN {X 30.883,Y -37.985,Z -55.943,A -90.000,B 90.000,C 0.000} C_DIS
LIN {X 31.036,Y -37.876,Z -55.788,A -90.000,B 90.000,C 0.000} C_DIS
LIN {X 31.163,Y -37.795,Z -55.671,A -90.000,B 90.000,C 0.000} C_DIS
LIN {X 31.223,Y -37.759,Z -55.622,A -90.000,B 90.000,C 0.000} C_DIS
LIN {X 31.269,Y -37.731,Z -55.589,A -90.000,B 90.000,C 0.000} C_DIS
LIN {X 31.427,Y -37.643,Z -55.485,A -90.000,B 90.000,C 0.000} C_DIS
LIN {X 31.489,Y -37.613,Z -55.449,A -90.000,B 90.000,C 0.000} C_DIS
LIN {X 31.518,Y -37.599,Z -55.435,A -90.000,B 90.000,C 0.000} C_DIS
LIN {X 31.598,Y -37.617,Z -55.143,A -90.000,B 90.000,C 0.000} C_DIS
LIN {X 31.642,Y -37.625,Z -54.992,A -90.000,B 90.000,C 0.000} C_DIS
LIN {X 31.665,Y -37.633,Z -54.908,A -90.000,B 90.000,C 0.000} C_DIS
LIN {X 31.762,Y -37.666,Z -54.578,A -90.000,B 90.000,C 0.000} C_DIS
LIN {X 31.807,Y -37.681,Z -54.433,A -90.000,B 90.000,C 0.000} C_DIS
LIN {X 31.929,Y -37.718,Z -54.086,A -90.000,B 90.000,C 0.000} C_DIS
LIN {X 32.010,Y -37.731,Z -53.899,A -90.000,B 90.000,C 0.000} C_DIS
LIN {X 32.044,Y -37.733,Z -53.814,A -90.000,B 90.000,C 0.000} C_DIS
LIN {X 32.094,Y -37.740,Z -53.695,A -90.000,B 90.000,C 0.000} C_DIS
LIN {X 32.174,Y -37.742,Z -53.539,A -90.000,B 90.000,C 0.000} C_DIS
LIN {X 32.273,Y -37.751,Z -53.327,A -90.000,B 90.000,C 0.000} C_DIS
LIN {X 32.405,Y -37.776,Z -53.076,A -90.000,B 90.000,C 0.000} C_DIS
LIN {X 32.509,Y -37.793,Z -52.888,A -90.000,B 90.000,C 0.000} C_DIS
LIN {X 32.596,Y -37.807,Z -52.746,A -90.000,B 90.000,C 0.000} C_DIS
LIN {X 32.728,Y -37.834,Z -52.544,A -90.000,B 90.000,C 0.000} C_DIS
LIN {X 32.861,Y -37.848,Z -52.365,A -90.000,B 90.000,C 0.000} C_DIS
LIN {X 33.058,Y -37.854,Z -52.089,A -90.000,B 90.000,C 0.000} C_DIS
LIN {X 33.150,Y -37.855,Z -51.973,A -90.000,B 90.000,C 0.000} C_DIS
LIN {X 33.406,Y -37.868,Z -51.662,A -90.000,B 90.000,C 0.000} C_DIS
LIN {X 33.524,Y -37.873,Z -51.536,A -90.000,B 90.000,C 0.000} C_DIS
LIN {X 33.678,Y -37.887,Z -51.380,A -90.000,B 90.000,C 0.000} C_DIS
LIN {X 33.816,Y -37.888,Z -51.258,A -90.000,B 90.000,C 0.000} C_DIS
LIN {X 33.998,Y -37.895,Z -51.103,A -90.000,B 90.000,C 0.000} C_DIS
LIN {X 34.075,Y -37.896,Z -51.042,A -90.000,B 90.000,C 0.000} C_DIS
LIN {X 34.214,Y -37.892,Z -50.925,A -90.000,B 90.000,C 0.000} C_DIS
LIN {X 34.417,Y -37.895,Z -50.745,A -90.000,B 90.000,C 0.000} C_DIS
LIN {X 34.541,Y -37.902,Z -50.643,A -90.000,B 90.000,C 0.000} C_DIS
LIN {X 34.889,Y -37.905,Z -50.401,A -90.000,B 90.000,C 0.000} C_DIS
LIN {X 35.030,Y -37.902,Z -50.322,A -90.000,B 90.000,C 0.000} C_DIS
LIN {X 35.237,Y -37.904,Z -50.213,A -90.000,B 90.000,C 0.000} C_DIS
LIN {X 35.377,Y -37.902,Z -50.143,A -90.000,B 90.000,C 0.000} C_DIS
LIN {X 35.543,Y -37.902,Z -50.065,A -90.000,B 90.000,C 0.000} C_DIS
LIN {X 35.593,Y -37.904,Z -50.040,A -90.000,B 90.000,C 0.000} C_DIS
LIN {X 35.950,Y -37.909,Z -49.862,A -90.000,B 90.000,C 0.000} C_DIS
LIN {X 36.190,Y -37.900,Z -49.757,A -90.000,B 90.000,C 0.000} C_DIS
LIN {X 36.348,Y -37.901,Z -49.695,A -90.000,B 90.000,C 0.000} C_DIS
LIN {X 36.583,Y -37.889,Z -49.621,A -90.000,B 90.000,C 0.000} C_DIS
LIN {X 36.746,Y -37.882,Z -49.572,A -90.000,B 90.000,C 0.000} C_DIS
LIN {X 36.845,Y -37.879,Z -49.550,A -90.000,B 90.000,C 0.000} C_DIS
LIN {X 37.273,Y -37.870,Z -49.461,A -90.000,B 90.000,C 0.000} C_DIS
LIN {X 37.613,Y -37.878,Z -49.393,A -90.000,B 90.000,C 0.000} C_DIS
LIN {X 38.026,Y -37.871,Z -49.329,A -90.000,B 90.000,C 0.000} C_DIS
LIN {X 38.214,Y -37.856,Z -49.312,A -90.000,B 90.000,C 0.000} C_DIS
LIN {X 38.435,Y -37.846,Z -49.299,A -90.000,B 90.000,C 0.000} C_DIS
LIN {X 38.677,Y -37.827,Z -49.294,A -90.000,B 90.000,C 0.000} C_DIS
LIN {X 38.800,Y -37.820,Z -49.294,A -90.000,B 90.000,C 0.000} C_DIS
LIN {X 39.293,Y -37.814,Z -49.311,A -90.000,B 90.000,C 0.000} C_DIS
LIN {X 39.982,Y -37.831,Z -49.353,A -90.000,B 90.000,C 0.000} C_DIS
LIN {X 40.408,Y -37.815,Z -49.408,A -90.000,B 90.000,C 0.000} C_DIS
LIN {X 40.644,Y -37.798,Z -49.454,A -90.000,B 90.000,C 0.000} C_DIS
LIN {X 40.879,Y -37.779,Z -49.502,A -90.000,B 90.000,C 0.000} C_DIS
LIN {X 41.007,Y -37.772,Z -49.532,A -90.000,B 90.000,C 0.000} C_DIS
LIN {X 41.293,Y -37.764,Z -49.604,A -90.000,B 90.000,C 0.000} C_DIS
LIN {X 41.418,Y -37.758,Z -49.638,A -90.000,B 90.000,C 0.000} C_DIS
LIN {X 41.536,Y -37.756,Z -49.673,A -90.000,B 90.000,C 0.000} C_DIS
LIN {X 41.765,Y -37.757,Z -49.744,A -90.000,B 90.000,C 0.000} C_DIS
LIN {X 41.993,Y -37.755,Z -49.821,A -90.000,B 90.000,C 0.000} C_DIS
LIN {X 42.655,Y -37.739,Z -50.061,A -90.000,B 90.000,C 0.000} C_DIS
LIN {X 43.241,Y -37.726,Z -50.279,A -90.000,B 90.000,C 0.000} C_DIS
LIN {X 43.856,Y -37.746,Z -50.499,A -90.000,B 90.000,C 0.000} C_DIS
LIN {X 44.248,Y -37.757,Z -50.644,A -90.000,B 90.000,C 0.000} C_DIS
LIN {X 44.364,Y -37.768,Z -50.675,A -90.000,B 90.000,C 0.000} C_DIS
LIN {X 44.595,Y -37.799,Z -50.745,A -90.000,B 90.000,C 0.000} C_DIS
LIN {X 44.844,Y -37.826,Z -50.821,A -90.000,B 90.000,C 0.000} C_DIS
LIN {X 45.181,Y -37.904,Z -50.878,A -90.000,B 90.000,C 0.000} C_DIS
LIN {X 45.326,Y -37.939,Z -50.904,A -90.000,B 90.000,C 0.000} C_DIS
LIN {X 45.550,Y -37.997,Z -50.946,A -90.000,B 90.000,C 0.000} C_DIS
LIN {X 45.633,Y -38.012,Z -50.954,A -90.000,B 90.000,C 0.000} C_DIS
LIN {X 46.052,Y -38.033,Z -50.913,A -90.000,B 90.000,C 0.000} C_DIS
LIN {X 46.633,Y -38.038,Z -50.826,A -90.000,B 90.000,C 0.000} C_DIS
LIN {X 47.141,Y -38.046,Z -50.746,A -90.000,B 90.000,C 0.000} C_DIS
LIN {X 47.423,Y -38.041,Z -50.711,A -90.000,B 90.000,C 0.000} C_DIS
LIN {X 47.540,Y -38.043,Z -50.700,A -90.000,B 90.000,C 0.000} C_DIS
LIN {X 47.828,Y -38.037,Z -50.682,A -90.000,B 90.000,C 0.000} C_DIS
LIN {X 47.991,Y -38.038,Z -50.677,A -90.000,B 90.000,C 0.000} C_DIS
LIN {X 48.262,Y -38.045,Z -50.672,A -90.000,B 90.000,C 0.000} C_DIS
LIN {X 48.819,Y -38.051,Z -50.656,A -90.000,B 90.000,C 0.000} C_DIS
LIN {X 49.297,Y -38.063,Z -50.636,A -90.000,B 90.000,C 0.000} C_DIS
LIN {X 49.588,Y -38.057,Z -50.635,A -90.000,B 90.000,C 0.000} C_DIS
LIN {X 49.698,Y -38.057,Z -50.637,A -90.000,B 90.000,C 0.000} C_DIS
LIN {X 50.090,Y -38.038,Z -50.674,A -90.000,B 90.000,C 0.000} C_DIS
LIN {X 50.227,Y -38.028,Z -50.696,A -90.000,B 90.000,C 0.000} C_DIS
LIN {X 50.653,Y -38.015,Z -50.787,A -90.000,B 90.000,C 0.000} C_DIS
LIN {X 50.815,Y -38.015,Z -50.827,A -90.000,B 90.000,C 0.000} C_DIS
LIN {X 51.296,Y -38.030,Z -50.960,A -90.000,B 90.000,C 0.000} C_DIS
LIN {X 51.769,Y -38.037,Z -51.084,A -90.000,B 90.000,C 0.000} C_DIS
LIN {X 52.116,Y -38.051,Z -51.167,A -90.000,B 90.000,C 0.000} C_DIS
LIN {X 52.505,Y -38.051,Z -51.273,A -90.000,B 90.000,C 0.000} C_DIS
LIN {X 52.653,Y -38.040,Z -51.323,A -90.000,B 90.000,C 0.000} C_DIS
LIN {X 52.874,Y -38.029,Z -51.403,A -90.000,B 90.000,C 0.000} C_DIS
LIN {X 52.987,Y -38.019,Z -51.449,A -90.000,B 90.000,C 0.000} C_DIS
LIN {X 53.157,Y -38.006,Z -51.519,A -90.000,B 90.000,C 0.000} C_DIS
LIN {X 53.242,Y -38.002,Z -51.559,A -90.000,B 90.000,C 0.000} C_DIS
LIN {X 53.590,Y -37.976,Z -51.752,A -90.000,B 90.000,C 0.000} C_DIS
LIN {X 53.702,Y -37.970,Z -51.819,A -90.000,B 90.000,C 0.000} C_DIS
LIN {X 54.071,Y -37.959,Z -52.048,A -90.000,B 90.000,C 0.000} C_DIS
LIN {X 54.180,Y -37.959,Z -52.119,A -90.000,B 90.000,C 0.000} C_DIS
LIN {X 55.432,Y -37.996,Z -52.983,A -90.000,B 90.000,C 0.000} C_DIS
LIN {X 55.575,Y -37.998,Z -53.078,A -90.000,B 90.000,C 0.000} C_DIS
LIN {X 55.760,Y -37.992,Z -53.210,A -90.000,B 90.000,C 0.000} C_DIS
LIN {X 55.914,Y -37.983,Z -53.323,A -90.000,B 90.000,C 0.000} C_DIS
LIN {X 56.175,Y -37.958,Z -53.528,A -90.000,B 90.000,C 0.000} C_DIS
LIN {X 56.538,Y -37.933,Z -53.826,A -90.000,B 90.000,C 0.000} C_DIS
LIN {X 56.659,Y -37.929,Z -53.931,A -90.000,B 90.000,C 0.000} C_DIS
LIN {X 56.968,Y -37.935,Z -54.219,A -90.000,B 90.000,C 0.000} C_DIS
LIN {X 57.367,Y -37.948,Z -54.601,A -90.000,B 90.000,C 0.000} C_DIS
LIN {X 57.938,Y -37.960,Z -55.155,A -90.000,B 90.000,C 0.000} C_DIS
LIN {X 58.315,Y -37.966,Z -55.523,A -90.000,B 90.000,C 0.000} C_DIS
LIN {X 58.544,Y -37.950,Z -55.772,A -90.000,B 90.000,C 0.000} C_DIS
LIN {X 58.946,Y -37.931,Z -56.199,A -90.000,B 90.000,C 0.000} C_DIS
LIN {X 59.104,Y -37.925,Z -56.370,A -90.000,B 90.000,C 0.000} C_DIS
LIN {X 59.145,Y -37.925,Z -56.418,A -90.000,B 90.000,C 0.000} C_DIS
LIN {X 59.481,Y -37.933,Z -56.817,A -90.000,B 90.000,C 0.000} C_DIS
LIN {X 59.621,Y -37.940,Z -56.988,A -90.000,B 90.000,C 0.000} C_DIS
LIN {X 60.115,Y -37.965,Z -57.597,A -90.000,B 90.000,C 0.000} C_DIS
LIN {X 60.400,Y -37.990,Z -57.968,A -90.000,B 90.000,C 0.000} C_DIS
LIN {X 60.611,Y -38.004,Z -58.251,A -90.000,B 90.000,C 0.000} C_DIS
LIN {X 61.015,Y -38.022,Z -58.812,A -90.000,B 90.000,C 0.000} C_DIS
LIN {X 61.394,Y -38.040,Z -59.342,A -90.000,B 90.000,C 0.000} C_DIS
LIN {X 61.937,Y -38.091,Z -60.151,A -90.000,B 90.000,C 0.000} C_DIS
LIN {X 62.337,Y -38.116,Z -60.771,A -90.000,B 90.000,C 0.000} C_DIS
LIN {X 62.554,Y -38.126,Z -61.112,A -90.000,B 90.000,C 0.000} C_DIS
LIN {X 62.815,Y -38.128,Z -61.536,A -90.000,B 90.000,C 0.000} C_DIS
LIN {X 62.875,Y -38.130,Z -61.639,A -90.000,B 90.000,C 0.000} C_DIS
LIN {X 63.209,Y -38.157,Z -62.249,A -90.000,B 90.000,C 0.000} C_DIS
LIN {X 63.678,Y -38.187,Z -63.079,A -90.000,B 90.000,C 0.000} C_DIS
LIN {X 64.176,Y -38.220,Z -63.968,A -90.000,B 90.000,C 0.000} C_DIS
LIN {X 64.225,Y -38.222,Z -64.059,A -90.000,B 90.000,C 0.000} C_DIS
LIN {X 64.403,Y -38.235,Z -64.375,A -90.000,B 90.000,C 0.000} C_DIS
LIN {X 64.808,Y -38.262,Z -65.101,A -90.000,B 90.000,C 0.000} C_DIS
LIN {X 64.858,Y -38.267,Z -65.195,A -90.000,B 90.000,C 0.000} C_DIS
LIN {X 65.384,Y -38.285,Z -66.092,A -90.000,B 90.000,C 0.000} C_DIS
LIN {X 65.744,Y -38.255,Z -66.586,A -90.000,B 90.000,C 0.000} C_DIS
LIN {X 66.020,Y -38.248,Z -66.949,A -90.000,B 90.000,C 0.000} C_DIS
LIN {X 66.249,Y -38.246,Z -67.259,A -90.000,B 90.000,C 0.000} C_DIS
LIN {X 66.331,Y -38.247,Z -67.376,A -90.000,B 90.000,C 0.000} C_DIS
LIN {X 66.722,Y -38.239,Z -67.903,A -90.000,B 90.000,C 0.000} C_DIS
LIN {X 66.960,Y -38.258,Z -68.201,A -90.000,B 90.000,C 0.000} C_DIS
LIN {X 67.263,Y -38.245,Z -68.498,A -90.000,B 90.000,C 0.000} C_DIS
LIN {X 67.517,Y -38.230,Z -68.751,A -90.000,B 90.000,C 0.000} C_DIS
LIN {X 67.581,Y -38.228,Z -68.813,A -90.000,B 90.000,C 0.000} C_DIS
LIN {X 67.778,Y -38.230,Z -69.008,A -90.000,B 90.000,C 0.000} C_DIS
LIN {X 67.858,Y -38.229,Z -69.089,A -90.000,B 90.000,C 0.000} C_DIS
LIN {X 67.945,Y -38.230,Z -69.182,A -90.000,B 90.000,C 0.000} C_DIS
LIN {X 68.347,Y -38.204,Z -69.548,A -90.000,B 90.000,C 0.000} C_DIS
LIN {X 68.439,Y -38.200,Z -69.637,A -90.000,B 90.000,C 0.000} C_DIS
LIN {X 68.793,Y -38.193,Z -69.996,A -90.000,B 90.000,C 0.000} C_DIS
LIN {X 69.110,Y -38.207,Z -70.298,A -90.000,B 90.000,C 0.000} C_DIS
LIN {X 69.277,Y -38.200,Z -70.430,A -90.000,B 90.000,C 0.000} C_DIS
LIN {X 69.796,Y -38.187,Z -70.865,A -90.000,B 90.000,C 0.000} C_DIS
LIN {X 70.321,Y -38.174,Z -71.305,A -90.000,B 90.000,C 0.000} C_DIS
LIN {X 70.670,Y -38.167,Z -71.621,A -90.000,B 90.000,C 0.000} C_DIS
LIN {X 71.022,Y -38.170,Z -71.933,A -90.000,B 90.000,C 0.000} C_DIS
LIN {X 71.466,Y -38.162,Z -72.307,A -90.000,B 90.000,C 0.000} C_DIS
LIN {X 72.148,Y -38.152,Z -72.887,A -90.000,B 90.000,C 0.000} C_DIS
LIN {X 72.664,Y -38.142,Z -73.329,A -90.000,B 90.000,C 0.000} C_DIS
LIN {X 73.225,Y -38.143,Z -73.833,A -90.000,B 90.000,C 0.000} C_DIS
LIN {X 73.455,Y -38.142,Z -74.041,A -90.000,B 90.000,C 0.000} C_DIS
LIN {X 73.568,Y -38.139,Z -74.146,A -90.000,B 90.000,C 0.000} C_DIS
LIN {X 73.660,Y -38.138,Z -74.236,A -90.000,B 90.000,C 0.000} C_DIS
LIN {X 73.987,Y -38.139,Z -74.569,A -90.000,B 90.000,C 0.000} C_DIS
LIN {X 74.127,Y -38.130,Z -74.693,A -90.000,B 90.000,C 0.000} C_DIS
LIN {X 74.260,Y -38.123,Z -74.815,A -90.000,B 90.000,C 0.000} C_DIS
LIN {X 74.736,Y -38.115,Z -75.285,A -90.000,B 90.000,C 0.000} C_DIS
LIN {X 74.873,Y -38.117,Z -75.434,A -90.000,B 90.000,C 0.000} C_DIS
LIN {X 74.957,Y -38.111,Z -75.518,A -90.000,B 90.000,C 0.000} C_DIS
LIN {X 75.036,Y -38.108,Z -75.601,A -90.000,B 90.000,C 0.000} C_DIS
LIN {X 75.491,Y -38.096,Z -76.105,A -90.000,B 90.000,C 0.000} C_DIS
LIN {X 75.538,Y -38.091,Z -76.150,A -90.000,B 90.000,C 0.000} C_DIS
LIN {X 75.897,Y -38.086,Z -76.486,A -90.000,B 90.000,C 0.000} C_DIS
LIN {X 76.075,Y -38.082,Z -76.654,A -90.000,B 90.000,C 0.000} C_DIS
LIN {X 76.214,Y -38.085,Z -76.799,A -90.000,B 90.000,C 0.000} C_DIS
LIN {X 76.345,Y -38.077,Z -76.921,A -90.000,B 90.000,C 0.000} C_DIS
LIN {X 76.599,Y -38.073,Z -77.175,A -90.000,B 90.000,C 0.000} C_DIS
LIN {X 76.809,Y -38.069,Z -77.331,A -90.000,B 90.000,C 0.000} C_DIS
LIN {X 76.900,Y -38.069,Z -77.402,A -90.000,B 90.000,C 0.000} C_DIS
LIN {X 76.997,Y -38.075,Z -77.479,A -90.000,B 90.000,C 0.000} C_DIS
LIN {X 77.134,Y -38.073,Z -77.571,A -90.000,B 90.000,C 0.000} C_DIS
LIN {X 77.217,Y -38.040,Z -77.581,A -90.000,B 90.000,C 0.000} C_DIS
LIN {X 77.242,Y -38.039,Z -77.577,A -90.000,B 90.000,C 0.000} C_DIS
LIN {X 77.390,Y -38.046,Z -77.547,A -90.000,B 90.000,C 0.000} C_DIS
LIN {X 77.517,Y -37.911,Z -77.363,A -90.000,B 90.000,C 0.000} C_DIS
LIN {X 77.547,Y -37.883,Z -77.324,A -90.000,B 90.000,C 0.000} C_DIS
LIN {X 77.685,Y -37.768,Z -77.157,A -90.000,B 90.000,C 0.000} C_DIS
LIN {X 77.792,Y -37.688,Z -77.039,A -90.000,B 90.000,C 0.000} C_DIS
LIN {X 77.990,Y -37.560,Z -76.854,A -90.000,B 90.000,C 0.000} C_DIS
LIN {X 78.013,Y -37.544,Z -76.563,A -90.000,B 90.000,C 0.000} C_DIS
LIN {X 78.026,Y -37.534,Z -76.259,A -90.000,B 90.000,C 0.000} C_DIS
LIN {X 78.043,Y -37.511,Z -75.784,A -90.000,B 90.000,C 0.000} C_DIS
LIN {X 78.065,Y -37.491,Z -75.463,A -90.000,B 90.000,C 0.000} C_DIS
LIN {X 78.084,Y -37.480,Z -75.004,A -90.000,B 90.000,C 0.000} C_DIS
LIN {X 78.095,Y -37.469,Z -74.713,A -90.000,B 90.000,C 0.000} C_DIS
LIN {X 78.140,Y -37.446,Z -74.079,A -90.000,B 90.000,C 0.000} C_DIS
LIN {X 78.206,Y -37.417,Z -73.294,A -90.000,B 90.000,C 0.000} C_DIS
LIN {X 78.220,Y -37.411,Z -73.082,A -90.000,B 90.000,C 0.000} C_DIS
LIN {X 78.267,Y -37.393,Z -72.584,A -90.000,B 90.000,C 0.000} C_DIS
LIN {X 78.334,Y -37.376,Z -71.987,A -90.000,B 90.000,C 0.000} C_DIS
LIN {X 78.424,Y -37.360,Z -71.445,A -90.000,B 90.000,C 0.000} C_DIS
LIN {X 78.467,Y -37.355,Z -71.197,A -90.000,B 90.000,C 0.000} C_DIS
LIN {X 78.514,Y -37.350,Z -70.974,A -90.000,B 90.000,C 0.000} C_DIS
LIN {X 78.585,Y -37.342,Z -70.650,A -90.000,B 90.000,C 0.000} C_DIS
LIN {X 78.676,Y -37.332,Z -70.342,A -90.000,B 90.000,C 0.000} C_DIS
LIN {X 78.795,Y -37.326,Z -69.942,A -90.000,B 90.000,C 0.000} C_DIS
LIN {X 79.033,Y -37.316,Z -69.224,A -90.000,B 90.000,C 0.000} C_DIS
LIN {X 79.189,Y -37.312,Z -68.772,A -90.000,B 90.000,C 0.000} C_DIS
LIN {X 79.783,Y -37.308,Z -67.277,A -90.000,B 90.000,C 0.000} C_DIS
LIN {X 79.809,Y -37.308,Z -67.211,A -90.000,B 90.000,C 0.000} C_DIS
LIN {X 79.808,Y -39.083,Z -67.215,A -90.000,B 90.000,C 0.000} C_DIS
LIN {X 79.811,Y -37.308,Z -67.205,A -90.000,B 90.000,C 0.000} C_DIS
LIN {X 79.816,Y -37.307,Z -67.192,A -90.000,B 90.000,C 0.000} C_DIS
LIN {X 79.848,Y -37.308,Z -67.130,A -90.000,B 90.000,C 0.000} C_DIS
LIN {X 79.894,Y -37.308,Z -67.025,A -90.000,B 90.000,C 0.000} C_DIS
LIN {X 79.894,Y -60.000,Z -67.025,A -90.000,B 90.000,C 0.000} C_DIS
LIN {X 89.627,Y -60.000,Z -54.009,A -90.000,B 90.000,C 0.000} C_DIS
LIN {X 89.627,Y -37.308,Z -54.009,A -90.000,B 90.000,C 0.000} C_DIS
LIN {X 89.714,Y -37.308,Z -53.929,A -90.000,B 90.000,C 0.000} C_DIS
LIN {X 89.714,Y -60.000,Z -53.929,A -90.000,B 90.000,C 0.000} C_DIS
LIN {X 97.312,Y -60.000,Z -47.248,A -90.000,B 90.000,C 0.000} C_DIS
LIN {X 97.312,Y -37.308,Z -47.248,A -90.000,B 90.000,C 0.000} C_DIS
LIN {X 97.468,Y -37.310,Z -47.096,A -90.000,B 90.000,C 0.000} C_DIS
LIN {X 97.648,Y -37.308,Z -46.921,A -90.000,B 90.000,C 0.000} C_DIS
LIN {X 97.818,Y -44.949,Z -46.756,A -90.000,B 90.000,C 0.000} C_DIS
LIN {X 97.899,Y -44.972,Z -46.677,A -90.000,B 90.000,C 0.000} C_DIS
LIN {X 97.978,Y -44.986,Z -46.601,A -90.000,B 90.000,C 0.000} C_DIS
LIN {X 98.127,Y -44.997,Z -46.457,A -90.000,B 90.000,C 0.000} C_DIS
LIN {X 98.266,Y -44.997,Z -46.322,A -90.000,B 90.000,C 0.000} C_DIS
LIN {X 98.732,Y -44.952,Z -45.873,A -90.000,B 90.000,C 0.000} C_DIS
LIN {X 99.066,Y -44.897,Z -45.551,A -90.000,B 90.000,C 0.000} C_DIS
